// TwinCAT 3 PLC project PLC_Framework_V2_00
// ProgramVersion: 3.1.4023.0
// libraries:
//   CAA Memory, * (CAA Technical Workgroup)
//   Tc2_Math, * (Beckhoff Automation GmbH)
//   Tc2_MC2, * (Beckhoff Automation GmbH)
//   Tc2_MC2_Drive, * (Beckhoff Automation GmbH)
//   Tc2_Standard, * (Beckhoff Automation GmbH)
//   Tc2_System, * (Beckhoff Automation GmbH)
//   Tc2_Utilities, * (Beckhoff Automation GmbH)
//   Tc3_Module, * (Beckhoff Automation GmbH)
// project tree:
//   / CheckBounds.TcPOU, CheckDivDInt.TcPOU, CheckDivLInt.TcPOU, CheckDivLReal.TcPOU, CheckDivReal.TcPOU, CheckLRangeSigned.TcPOU, CheckLRangeUnsigned.TcPOU, CheckPointer.TcPOU, CheckRangeSigned.TcPOU, CheckRangeUnsigned.TcPOU, PlcTask.TcTTO
//   GVLs/ GVL_Module.TcGVL, GVL_Constant.TcGVL, GVL_Standard.TcGVL
//   POUs/ MAIN.TcPOU
//   Standard/ CallStandard.TcPOU, CallStandardModule.TcPOU
//   Standard/ENUM/ ENUM_CarrierPos.TcDUT, ENUM_ExecState.TcDUT, ENUM_NgReason.TcDUT, ENUM_ProductState.TcDUT, ENUM_StationCommand.TcDUT, ENUM_UnitState.TcDUT
//   Standard/FUN/ FUN_AryBitCount_RD.TcPOU, FUN_AryBitOnNum_RD.TcPOU, FUN_AryToLword_RD.TcPOU, FUN_AryToWord_RD.TcPOU, FUN_TimeToDate_RD.TcPOU, FUN_UpdateLeftSidebar_RD.TcPOU, FUN_WordToAry.TcPOU, F_Sum.TcPOU
//   Standard/Module/Connector/Termininal/ FB_Terminal2_RD.TcPOU, FB_Terminal_RD.TcPOU, UDT_TerminalData_RD.TcDUT, UDT_TerminalHmi_RD.TcDUT, UDT_TerminalMessage_RD.TcDUT, UDT_TerminalVar_RD.TcDUT, UDT_Terminal_RD.TcDUT
//   Standard/Module/FAKRA/BraidFlaring/ FB_BraidFlaring_RD.TcPOU, UDT_BraidFlaring_RD.TcDUT, UDT_Data_BraidFlaring_RD.TcDUT, UDT_Hmi_BraidFlaring_RD.TcDUT, UDT_Imm_BraidFlaring_RD.TcDUT, UDT_Parameters_BraidFlaring_RD.TcDUT
//   Standard/Module/FAKRA/Crimping/ FB_Crimping_RD.TcPOU, UDT_Crimping_RD.TcDUT, UDT_Data_Crimping_RD.TcDUT, UDT_Hmi_Crimping_RD.TcDUT, UDT_Imm_Crimping_RD.TcDUT, UDT_Parameters_Crimping_RD.TcDUT
//   Standard/Module/FAKRA/JacketStripping/ FB_JacketStripping_RD.TcPOU, UDT_CriticalProcessParameters_JacketStripping_RD.TcDUT, UDT_Data_JacketStripping_RD.TcDUT, UDT_Hmi_JacketStripping_RD.TcDUT, UDT_Imm_JacketStripping_RD.TcDUT, UDT_JacketStripping_RD.TcDUT
//   Standard/Public/00 System/ FB_Blinker_RD.TcPOU, FB_GetPlcClock.TcPOU, UDT_PlcStatus_RD.TcDUT, UDT_ProgramStatus_RD.TcDUT, UDT_System_RD.TcDUT
//   Standard/Public/01 Machine/ FB_Machine_RD.TcPOU, UDT_MachineHmi_RD.TcDUT, UDT_MachineReport_RD.TcDUT, UDT_MachineSidebar_RD.TcDUT, UDT_Machine_RD.TcDUT
//   Standard/Public/02 Station/ FB_Station_RD.TcPOU, UDT_FlowHmi_RD.TcDUT, UDT_Flow_RD.TcDUT, UDT_StationHmi_RD.TcDUT, UDT_StationMessage_RD.TcDUT, UDT_StationReport_RD.TcDUT, UDT_StationSidebar_RD.TcDUT, UDT_Station_RD.TcDUT
//   Standard/Public/03 HMI/ UDT_RightSidebar_RD.TcDUT, FB_GetPageSerialNo_RD.TcPOU, FB_GetPlcClock_RD.TcPOU, FB_Hmi_RD.TcPOU, FB_IV3_G120_RD.TcPOU, FB_Tben_L5_4Rfid_RD.TcPOU, FB_TurnPages_RD.TcPOU, FB_UpdateAxisHmi_RD.TcPOU, FB_UpdateCycleTimeHmi_RD.TcPOU, FB_UpdateInsertHmi_RD.TcPOU, FB_UpdateProduceHmi_RD.TcPOU, UDT_Clock_RD.TcDUT, UDT_CycleTimeHmi_RD.TcDUT, UDT_DayTime_RD.TcDUT, UDT_Hmi_RD.TcDUT, UDT_HmiButton_RD.TcDUT, UDT_LeftSidebar_RD.TcDUT, UDT_TurnPages_RD.TcDUT
//   Standard/Public/06 Produce/ FB_Produce_RD.TcPOU, FB_Produce.TcPOU, UDT_BadData_RD.TcDUT, UDT_BadHmi_RD.TcDUT, UDT_BadVar_RD.TcDUT, UDT_ProduceDataRecord_RD.TcDUT, UDT_ProduceData_RD.TcDUT, UDT_ProduceHmi_RD.TcDUT, UDT_ProduceVar_RD.TcDUT
//   Standard/Public/08 WearPart/ FB_WearPart.TcPOU, UDT_WearPartData_RD.TcDUT, UDT_WearPartHmi_RD.TcDUT, UDT_WearPartVar_RD.TcDUT
//   Standard/Public/11 Oee/ FB_Oee_RD.TcPOU, UDT_OeeData_RD.TcDUT, UDT_OeeHmi_RD.TcDUT, UDT_OeeVar_RD.TcDUT
//   Standard/Unit/00 General/ FB_Click_RD.TcPOU
//   Standard/Unit/03 Estop/ FB_Estop_RD.TcPOU, UDT_Estop_RD.TcDUT
//   Standard/Unit/04 SafetyDoor/ FB_SafetyDoor_RD.TcPOU, UDT_SafetyDoor_RD.TcDUT
//   Standard/Unit/05 Cylinder/ FB_Cylinder_RD.TcPOU, UDT_CylinderData_RD.TcDUT, UDT_CylinderHmi_RD.TcDUT, UDT_CylinderMessage_RD.TcDUT, UDT_CylinderVar_RD.TcDUT
//   Standard/Unit/06 Axis/ FB_Axis_RD.TcPOU, FB_ModuloCalculate_RD.TcPOU, FB_NCI.TcPOU, UDT_AxisData_RD.TcDUT, UDT_AxisHmi_RD.TcDUT, UDT_AxisMessage_RD.TcDUT, UDT_AxisVar_RD.TcDUT, UDT_ModuloProperty_RD.TcDUT
//   Standard/Unit/07 Sensor/ FB_Sensor_RD.TcPOU, UDT_SensorData_RD.TcDUT, UDT_SensorHmi_RD.TcDUT, UDT_SensorVar_RD.TcDUT
//   Standard/Unit/08 Motor/ FB_Motor_RD.TcPOU, UDT_MotorData_RD.TcDUT, UDT_MotorHmi_RD.TcDUT, UDT_MotorVar_RD.TcDUT
//   Standard/Unit/11 KeyenceScan/ FB_KeyenceScan_RD.TcPOU, UDT_KeyenceScanData_RD.TcDUT, UDT_KeyenceScanHmi_RD.TcDUT, UDT_KeyenceScanVar_RD.TcDUT
//   Standard/Unit/12 Delay/ FB_Delay_RD.TcPOU, UDT_DelayData_RD.TcDUT, UDT_DelayHmi_RD.TcDUT, UDT_DelayVar_RD.TcDUT
//   Standard/Unit/13 Valve/ FB_Valve_RD.TcPOU, UDT_ValveData_RD.TcDUT, UDT_ValveHmi_RD.TcDUT, UDT_ValveVar_RD.TcDUT
//   Standard/Unit/40 RackFeeder/ FB_RackFeeder_RD.TcPOU, UDT_RackFeederData_RD.TcDUT, UDT_RackFeederHmi_RD.TcDUT, UDT_RackFeederInput_RD.TcDUT, UDT_RackFeederOutput_RD.TcDUT, UDT_RackFeederVar_RD.TcDUT, UDT_RackFeedMessage_RD.TcDUT

CONFIGURATION PLC_Framework_V2_00
    RESOURCE PLC ON TwinCAT3
        TASK PlcTask(INTERVAL := T#10ms, PRIORITY := 20);
        PROGRAM MAIN WITH PlcTask : MAIN;
    END_RESOURCE
END_CONFIGURATION

// ---- Standard/ENUM/ENUM_CarrierPos.TcDUT
TYPE ENUM_CarrierPos :
(
	Left 	:= 1,
	Right 	:= 2
)UINT;
END_TYPE

// ---- Standard/ENUM/ENUM_ExecState.TcDUT
{attribute 'qualified_only'}
{attribute 'strict'}
TYPE ENUM_ExecState :
(
	NOT_READY := 1,
  READY :=2,
  RUNNING :=3,
  DONE :=4,
  CANCEL :=5,
  INIT := 6,
  ERROR :=7

);
END_TYPE

// ---- Standard/ENUM/ENUM_NgReason.TcDUT
{attribute 'qualified_only'}
{attribute 'strict'}
TYPE ENUM_NgReason :
(
	CrimpNoCable :=1,
	CrimpNg,
	CrimpInterrupted,
	LastReason
);
END_TYPE

// ---- Standard/ENUM/ENUM_ProductState.TcDUT
{attribute 'qualified_only'}
{attribute 'strict'}
TYPE ENUM_ProductState :
(
	Empty:=0,					//无产品
	Good:=1,					//良品
	Bad:=2,						//不良品
	New:=3,						//新产品
	Sample:=4					//送检样品
);
END_TYPE

// ---- Standard/ENUM/ENUM_StationCommand.TcDUT
{attribute 'qualified_only'}
{attribute 'strict'}
TYPE ENUM_StationCommand :
(
  	
    INIT :=1,
    START := 2,
    STOP :=3,
    PAUSE := 4
    
    
  
);
END_TYPE

// ---- Standard/ENUM/ENUM_UnitState.TcDUT
{attribute 'qualified_only'}
{attribute 'strict'}
TYPE ENUM_UnitState :
(
  
	DISABLED := 1,
  OPERATIONAL :=2,
  STANDBY :=3,
  UNKNOWN :=4

);
END_TYPE

// ---- Standard/Module/Connector/Termininal/UDT_TerminalData_RD.TcDUT
TYPE UDT_TerminalData_RD :
STRUCT
timeout           : TIME; //对端子超时
terminalSensor    : UDT_SensorData_RD; //端子有无感应
coverSensor       : UDT_SensorData_RD; //盖板感应
pinSensor         : UDT_SensorData_RD; //对Pin感应
END_STRUCT
END_TYPE

// ---- Standard/Module/Connector/Termininal/UDT_TerminalHmi_RD.TcDUT
TYPE UDT_TerminalHmi_RD :
STRUCT
terminalSensor    : UDT_SensorHmi_RD; //端子有无感应
coverSensor       : UDT_SensorHmi_RD; //盖板感应
pinSensor         : UDT_SensorHmi_RD; //对Pin感应
hmi               : BOOL; //对端子Hmi
manual            : BOOL; //对端子手动执行
forbidIcon        : BOOL; //禁止图标
display           : BOOL; //显示
ready             : BOOL; //对端子准备就绪
busy              : BOOL; //对端子中
done              : BOOL; //对端子完成
subDisplay        : BOOL; //子画面显示
number            : INT; //编号
flowStep          : INT; //流程步
status            : INT; //状态
timeout           : DINT; //对端子超时
END_STRUCT
END_TYPE

// ---- Standard/Module/Connector/Termininal/UDT_TerminalMessage_RD.TcDUT
TYPE UDT_TerminalMessage_RD :
STRUCT
timeoutAlarm       : BOOL; //对端子超时报警
lackTerminalAlarm  : BOOL; //缺端子报警
coverAlarm         : BOOL; //盖板未检测到报警
alarming           : BOOL; //报警
END_STRUCT
END_TYPE

// ---- Standard/Module/Connector/Termininal/UDT_TerminalVar_RD.TcDUT
TYPE UDT_TerminalVar_RD :
STRUCT
terminalSensor       : UDT_SensorVar_RD; //端子有无感应
coverSensor          : UDT_SensorVar_RD; //盖板感应
pinSensor            : UDT_SensorVar_RD; //对Pin感应
disable              : BOOL; //屏蔽
hmi                  : BOOL; //对端子Hmi
manual               : BOOL; //对端子手动执行
auto                 : BOOL; //对端子自动执行
forbidIcon           : BOOL; //禁止图标
camAxisEnable        : BOOL; //插针凸轮轴启用
cutEnable            : BOOL; //裁切端子启用
running              : BOOL; //对端子运行中
ready                : BOOL; //对端子准备就绪
busy                 : BOOL; //对端子中
permit               : BOOL; //对端子条件
allow                : BOOL; //对端子可动作
done                 : BOOL; //对端子完成
faile                : BOOL; //对端子失败
timeoutAlarm         : BOOL; //对端子超时报警
lackTerminalAlarm    : BOOL; //缺端子报警
coverAlarm           : BOOL; //盖板未检测到报警
lackTerminalAutoTip  : BOOL; //缺端子自动提示
coverAutoTip         : BOOL; //盖板未检测到自动提示
alarming             : BOOL; //报警中
manualTip            : BOOL; //手动提示
autoTip              : BOOL; //自动提示
flowStep             : UINT; //流程步
status               : UINT; //状态
camAxisNo            : UINT; //凸轮轴
sendAxisNo           : UINT; //送端子轴
stationNo            : UINT; //所属工站编号
serialNo             : UINT; //HMI显示序号
END_STRUCT
END_TYPE

// ---- Standard/Module/Connector/Termininal/UDT_Terminal_RD.TcDUT
TYPE UDT_Terminal_RD :
STRUCT
send1Finish     : BOOL; //上进端子完成
send2Finish     : BOOL; //下进端子完成
send1Auto       : BOOL; //上进端子自动
send2Auto       : BOOL; //下进端子自动
END_STRUCT
END_TYPE

// ---- Standard/Module/FAKRA/BraidFlaring/UDT_BraidFlaring_RD.TcDUT
TYPE UDT_BraidFlaring_RD :
STRUCT
  
Imm : UDT_Imm_BraidFlaring_RD;
Message : UDT_StationMessage_RD;
Hmi : UDT_Hmi_BraidFlaring_RD;

UnitState : INT;	//DISABLED := 1,OPERATIONAL :=2,STANDBY :=3,UNKNOWN :=4
Command :INT; //INIT :=1,START := 2,STOP :=3,PAUSE := 4
CommandState : INT ; 	//NOT_READY := 1,READY :=2,RUNNING :=3,DONE :=4,CANCEL :=5,INIT := 6,ERROR :=7

END_STRUCT
END_TYPE

// ---- Standard/Module/FAKRA/BraidFlaring/UDT_Data_BraidFlaring_RD.TcDUT
TYPE UDT_Data_BraidFlaring_RD :
STRUCT
  
  gripCyl:UDT_CylinderData_RD;
  jackCyl:UDT_CylinderData_RD;
  pushCyl:UDT_CylinderData_RD;
  fixCyl:UDT_CylinderData_RD;
  stepFixCyl:UDT_CylinderData_RD;
  blow:UDT_CylinderData_RD;
  vacuum:UDT_CylinderData_RD;
  
  transferAxis : UDT_AxisData_RD;
  rotateAxis : UDT_AxisData_RD; 
  
  badDetectData :UDT_BadData_RD;//1227
  
  CPP : UDT_Parameters_BraidFlaring_RD;

END_STRUCT
END_TYPE

// ---- Standard/Module/FAKRA/BraidFlaring/UDT_Hmi_BraidFlaring_RD.TcDUT
TYPE UDT_Hmi_BraidFlaring_RD :
STRUCT

gripCyl:UDT_CylinderHmi_RD;
jackCyl:UDT_CylinderHmi_RD;
pushCyl:UDT_CylinderHmi_RD;
fixCyl:UDT_CylinderHmi_RD;
stepFixCyl:UDT_CylinderHmi_RD;
blow:UDT_CylinderHmi_RD;
vacuum:UDT_CylinderHmi_RD;

transferAxis : UDT_AxisHmi_RD; 
rotateAxis : UDT_AxisHmi_RD;

badDetect:UDT_BadHmi_RD;// 1227

station : UDT_StationHmi_RD;

END_STRUCT
END_TYPE

// ---- Standard/Module/FAKRA/BraidFlaring/UDT_Imm_BraidFlaring_RD.TcDUT
TYPE UDT_Imm_BraidFlaring_RD :
STRUCT
  
//公共接口
 Machine_eStop : BOOL;
 Machine_safety : BOOL;
 Machine_airOn : BOOL;
 Machine_allDoorClosed : BOOL;
 Machine_manualMode : BOOL; 
 Machine_autoMode : BOOL;
 Machine_reset :BOOL;
 Machine_stopping :BOOL;
 Machine_paused: BOOL;
 Machine_running :BOOL;

 
 //模组参数输入
 
 carrierNum		: UINT;	//载座编号（INPUT）
 carrierInPos : BOOL; //载座到位（INPUT）
 carrierPos :UINT; //载座位置（左1/右2）（INPUT）
 carrierState:UINT;//载座状态    //1227
 stationCanRun :BOOL;//模组动作条件（INPUT）
 
 //模组参数输出
 stationDone :BOOL;//模组完成（OUTPUT）
 carrierFree :BOOL;//载座不干涉（OUTPUT）
 carrierLeftProductState :INT; //左载座产品状态（OUTPUT）
 carrierRightProductState :INT;//右载座产品状态（OUTPUT）
 allObjectInitPos:BOOL;//所有部件在初始位置（OUTPUT）

 
END_STRUCT
END_TYPE

// ---- Standard/Module/FAKRA/BraidFlaring/UDT_Parameters_BraidFlaring_RD.TcDUT
TYPE UDT_Parameters_BraidFlaring_RD :
STRUCT
	clipEnable						: ARRAY [1..5] OF BOOL;
	transferAxisClipPosOffset		: ARRAY [1..5] OF REAL;
	rotateAxisClipPosOffset		    : ARRAY [1..5] OF REAL;
	transferAxisPushStartPosOffset	: REAL;
	transferAxisPushEndPosOffset	: REAL;
	rotateAxisPushPosOffset		    : REAL;
	rotateAxisBasePos				: REAL;
	transferAxisBasePos			    : REAL;
	override :INT;
END_STRUCT
END_TYPE

// ---- Standard/Module/FAKRA/Crimping/UDT_Crimping_RD.TcDUT
TYPE UDT_Crimping_RD :
STRUCT
  
Imm : UDT_Imm_Crimping_RD;
Message : UDT_StationMessage_RD;
Hmi : UDT_Hmi_Crimping_RD;

UnitState : INT;	//DISABLED := 1,OPERATIONAL :=2,STANDBY :=3,UNKNOWN :=4
Command :INT; //INIT :=1,START := 2,STOP :=3,PAUSE := 4
CommandState : INT ; 	//NOT_READY := 1,READY :=2,RUNNING :=3,DONE :=4,CANCEL :=5,INIT := 6,ERROR :=7

END_STRUCT
END_TYPE

// ---- Standard/Module/FAKRA/Crimping/UDT_Data_Crimping_RD.TcDUT
TYPE UDT_Data_Crimping_RD :
STRUCT
  
  gripCyl:UDT_CylinderData_RD;
  jack1Cyl:UDT_CylinderData_RD;
  jack2Cyl:UDT_CylinderData_RD;
  cutCyl:UDT_CylinderData_RD;
  feedCyl:UDT_CylinderData_RD;
  changeCyl:UDT_CylinderData_RD;
  fixCyl:UDT_CylinderData_RD;
  stepFixCyl:UDT_CylinderData_RD;
  carrierHold1Cyl:UDT_CylinderData_RD;
  carrierHold2Cyl:UDT_CylinderData_RD;
  jack3Cyl:UDT_CylinderData_RD;
  blow:UDT_CylinderData_RD;
  
  transferAxis : UDT_AxisData_RD; 
  crimpAxis : UDT_AxisData_RD;  
  
  rackFeeder:UDT_RackFeederData_RD;
  
  produceData:UDT_ProduceData_RD;
  badData: ARRAY[0..ENUM_NgReason.CrimpNg] OF UDT_BadData_RD;
  lastProduce:UDT_ProduceDataRecord_RD;
  
  CPP : UDT_Parameters_Crimping_RD;
  
  wearPart1 : UDT_WearPartData_RD;
  wearPart2 : UDT_WearPartData_RD;
 
  cableCheckSensorDisabled            : BOOL;
  terminalCheckSensorDisabled         : BOOL;
  terminalReiveCheckSensorDisabled    : BOOL;
  crimpHomeCheckSensorDisabled        : BOOL;
  oesDisabled                         : BOOL;  
  
END_STRUCT
END_TYPE

// ---- Standard/Module/FAKRA/Crimping/UDT_Hmi_Crimping_RD.TcDUT
TYPE UDT_Hmi_Crimping_RD :
STRUCT

gripCyl:UDT_CylinderHmi_RD;
jack1Cyl:UDT_CylinderHmi_RD;
jack2Cyl:UDT_CylinderHmi_RD;
cutCyl:UDT_CylinderHmi_RD;
feedCyl:UDT_CylinderHmi_RD;
changeCyl:UDT_CylinderHmi_RD;
fixCyl:UDT_CylinderHmi_RD;
stepFixCyl:UDT_CylinderHmi_RD;
carrierHold1Cyl:UDT_CylinderHmi_RD;
carrierHold2Cyl:UDT_CylinderHmi_RD;  
jack3Cyl:UDT_CylinderHmi_RD;
blow:UDT_CylinderHmi_RD; 

transferAxis : UDT_AxisHmi_RD; 
crimpAxis : UDT_AxisHmi_RD;

rackFeeder:UDT_RackFeederHmi_RD;

bad:UDT_BadHmi_RD;
produce:UDT_ProduceHmi_RD;

station : UDT_StationHmi_RD;

END_STRUCT
END_TYPE

// ---- Standard/Module/FAKRA/Crimping/UDT_Imm_Crimping_RD.TcDUT
TYPE UDT_Imm_Crimping_RD :
STRUCT
  
//公共接口
 Machine_eStop : BOOL;
 Machine_safety : BOOL;
 Machine_airOn : BOOL;
 Machine_allDoorClosed : BOOL;
 Machine_manualMode : BOOL; 
 Machine_autoMode : BOOL;
 Machine_reset :BOOL;
 Machine_stopping :BOOL;
 Machine_paused: BOOL;
 Machine_running :BOOL;

 
 //模组参数输入
 
 carrierNum		: UINT;	//载座编号（INPUT）
 carrierInPos : BOOL; //载座到位（INPUT）
 carrierPos :UINT; //载座位置（左1/右2）（INPUT）
 carrierState:UINT;//载座状态    //1227
 stationCanRun :BOOL;//模组动作条件（INPUT）
 
 //模组参数输出
 stationDone :BOOL;//模组完成（OUTPUT）
 carrierFree :BOOL;//载座不干涉（OUTPUT）
 carrierLeftProductState :INT; //左载座产品状态（OUTPUT）
 carrierRightProductState :INT;//右载座产品状态（OUTPUT）
 allObjectInitPos:BOOL;//所有部件在初始位置（OUTPUT）

 
END_STRUCT
END_TYPE

// ---- Standard/Module/FAKRA/Crimping/UDT_Parameters_Crimping_RD.TcDUT
TYPE UDT_Parameters_Crimping_RD :
STRUCT
	override :INT;
END_STRUCT
END_TYPE

// ---- Standard/Module/FAKRA/JacketStripping/UDT_CriticalProcessParameters_JacketStripping_RD.TcDUT
TYPE UDT_CriticalProcessParameters_JacketStripping_RD :
STRUCT
  
  blowTime :UDINT;
  firstCutTime :UDINT;
  firstOpenTime :UDINT;
  SecondCutTime :UDINT;
  secondOpenTime:UDINT;
  secondCutEnable	:BOOL;
  thirdCutTime	:UDINT;
  thirdOpenTime	:UDINT;
  thirdCutEnable	:BOOL;
  fourthCutTime	:UDINT;
  fourthOpenTime:	UDINT;
  fourthCutEnable	:BOOL;
  fifthCutTime	:UDINT;
  fifthOpenTime	:UDINT;
  fifthCutEnable	:BOOL;
  override :INT;
  
END_STRUCT
END_TYPE

// ---- Standard/Module/FAKRA/JacketStripping/UDT_Data_JacketStripping_RD.TcDUT
TYPE UDT_Data_JacketStripping_RD :
STRUCT
  
  gripCyl:UDT_CylinderData_RD;
  jackCyl:UDT_CylinderData_RD;
  fixCyl:UDT_CylinderData_RD;
  stepFixCyl:UDT_CylinderData_RD;
  blow:UDT_CylinderData_RD; 
  
  transferAxis : UDT_AxisData_RD; 
  cutAxis : UDT_AxisData_RD;  
  rotateAxis : UDT_AxisData_RD; 
  
  CPP : UDT_CriticalProcessParameters_JacketStripping_RD;
  
  wearPart : UDT_WearPartData_RD;
 
  
  
END_STRUCT
END_TYPE

// ---- Standard/Module/FAKRA/JacketStripping/UDT_Hmi_JacketStripping_RD.TcDUT
TYPE UDT_Hmi_JacketStripping_RD :
STRUCT
  
gripCyl : UDT_CylinderHmi_RD;
jackCyl :UDT_CylinderHmi_RD;
fixCyl  :UDT_CylinderHmi_RD;
stepFixCyl:UDT_CylinderHmi_RD; 
blow    :UDT_CylinderHmi_RD;

rotateAxis : UDT_AxisHmi_RD; 
cutAxis : UDT_AxisHmi_RD; 
transferAxis : UDT_AxisHmi_RD;

station : UDT_StationHmi_RD;

END_STRUCT
END_TYPE

// ---- Standard/Module/FAKRA/JacketStripping/UDT_Imm_JacketStripping_RD.TcDUT
TYPE UDT_Imm_JacketStripping_RD :
STRUCT
  
//公共接口（由外部机台输入）
 machine_eStop : BOOL;
 machine_safety : BOOL;
 machine_airOn : BOOL;
 machine_allDoorClosed : BOOL;
 machine_manualMode : BOOL; 
 machine_autoMode : BOOL;
 
 machine_running :BOOL;
 machine_stopping :BOOL;
 machine_initing :BOOL;
 machine_pause :BOOL;
 machine_reset :BOOL;

 //模组参数输入
 
 carrierNum		: UINT;	//载座编号（INPUT）
 carrierInPos : BOOL; //载座到位（INPUT）
 carrierPos :UINT; //载座位置（左1/右2）（INPUT）
 stationCanRun :BOOL;//模组动作条件（INPUT）

 
 //模组参数输出
 
 stationAlarming :BOOL;//模组报警中（OUTPUT）
 stationRunning :BOOL;//模组运行中（OUTPUT）
 stationInitDone :BOOL;//模组初始化完成（Output）
 stationDone :BOOL;//模组完成（OUTPUT）
 carrierFree :BOOL;//载座不干涉（OUTPUT）
 carrierLeftProductState :INT; //左载座产品状态（OUTPUT）
 carrierRightProductState :INT;//右载座产品状态（OUTPUT）
 allObjectInitPos:BOOL;//所有部件在初始位置（OUTPUT）
 
END_STRUCT
END_TYPE

// ---- Standard/Module/FAKRA/JacketStripping/UDT_JacketStripping_RD.TcDUT
TYPE UDT_JacketStripping_RD :
STRUCT
  
Imm : UDT_Imm_JacketStripping_RD;
Message : UDT_StationMessage_RD;
Hmi : UDT_Hmi_JacketStripping_RD;

UnitState : INT;	//DISABLED := 1,OPERATIONAL :=2,STANDBY :=3,UNKNOWN :=4
Command :INT; //INIT :=1,START := 2,STOP :=3,PAUSE := 4
CommandState : INT ; 	//NOT_READY := 1,READY :=2,RUNNING :=3,DONE :=4,CANCEL :=5,INIT := 6,ERROR :=7


END_STRUCT
END_TYPE

// ---- Standard/Public/00 System/UDT_PlcStatus_RD.TcDUT
TYPE UDT_PlcStatus_RD :
STRUCT
  
cycleTime : TIME; // 周期时间
maxCycleTime : Time; // 最长循环时间
minCycleTime : Time; // 最短循环时间
systemClock : DATE_AND_TIME; // 系统时钟
localClock : DATE_AND_TIME; // 本地时钟
status : Int; // CPU运行状态

END_STRUCT
END_TYPE

// ---- Standard/Public/00 System/UDT_ProgramStatus_RD.TcDUT
TYPE UDT_ProgramStatus_RD :
STRUCT
 
error : BOOL; // 有错误
errorID : Word; // 错误代码
errorText : String[100]; // 错误文本信息
warning : Bool; // 有警告
warnID : Word; // 警告代码
warnText : String[100]; // 警告文本信息
  
END_STRUCT
END_TYPE

// ---- Standard/Public/00 System/UDT_System_RD.TcDUT
TYPE UDT_System_RD :
STRUCT
clock	: UDT_Clock_RD;
plcStatus :	UDT_PlcStatus_RD;				
programStatus	: UDT_ProgramStatus_RD;
 
END_STRUCT
END_TYPE

// ---- Standard/Public/01 Machine/UDT_MachineHmi_RD.TcDUT
TYPE UDT_MachineHmi_RD :
STRUCT
eStop : BOOL; //急停
airOn : BOOL; //气压
allDoorClosed : BOOL; //安全门
ready : Bool; //准备就绪
running : Bool; //运行中
alarming : Bool; //报警中
paused : Bool; //暂停中
stopping : Bool; //停止中
tipReset : Bool; // 提示复位
initConfirm : Bool; // 整机初始化确认
emptyConfirm : Bool; // 清料确认
emptyhmi : Bool; // 清料hmi
emptying : Bool; // 清料中
emptyDone : Bool; // 清料完成
dummying : Bool; // 点检中
dummyDone : Bool; // 点检完成
dryRun : Bool; // 空跑
startButtonLight : Bool; // 启动按钮指示灯
stopButtonLight : Bool; // 停止按钮指示灯
resetButtonLight : Bool; // 复位按钮指示灯
pauseButtonLight : Bool; // 暂停按钮指示灯
initButtonLight : Bool; // 初始化按钮指示灯
starthmi : Bool; // 启动hmi
stophmi : Bool; // 停止hmi
resethmi : Bool; // 复位hmi
pausehmi : Bool; // 暂停hmi
inithmi : Bool; // 整机初始化hmi
manualModehmi : Bool; // 手动模式hmi
autoModehmi : Bool; // 自动模式hmi
jogModehmi : Bool; // 寸动模式hmi
setupModehmi : Bool; // 调试模式hmi
lampTesthmi : Bool; // 指示灯测试hmi
floodlighthmi : Bool; // 照明灯光打开hmi
alarmTopBarDisplay : Bool; // 报警顶栏显示
actAlarmTimes : UInt; // 当前发生报警条数
status : UInt; // 整机状态显示
initStatus : UInt; // 整机初始化状态显示
mode : UInt; // 操作模式
haveControlhmiNo : Int; // 当前拥有该机器控制权的hmi编号
requestControlhmiNo : Int; // 请求该机器控制权的hmi编号
requestCountdown : Int; // hmi请求控制权倒计时
actLanguage : Int; // 当前使用语言
mainScreenNo : Int; // 主画面编号
popup : Int; // 触摸屏弹窗
flow : Array[0..7] of UDT_FlowHmi_RD; // 流程
sidebar : UDT_LeftSidebar_RD; //
number : Int; // 机器编号
  
END_STRUCT
END_TYPE

// ---- Standard/Public/01 Machine/UDT_MachineReport_RD.TcDUT
TYPE UDT_MachineReport_RD :
STRUCT
alarming : BOOL; // 其它报警中
manualTip : Bool; // 其它手动提示
autoTip : Bool; // 其它自动提示
alarmCanReset : Bool; // 报警可复位
notSafetyDoors : Bool; // 安全门未就绪
notEstops : Bool; // 急停未就绪
stationAlarming : Bool; // 工站报警中
stationManualTip : Bool; // 工站手动提示
stationAutoTip : Bool; // 工站自动提示
stationNotInitDone : Bool; // 工站初始化未完成

END_STRUCT
END_TYPE

// ---- Standard/Public/01 Machine/UDT_MachineSidebar_RD.TcDUT
TYPE UDT_MachineSidebar_RD :
STRUCT
typeData : ARRAY[0..31] OF INT; // 按钮类型
status : ARRAY[0..31] OF Bool; // 按钮状态
click : ARRAY[0..31] OF Bool; // 按钮操作 
END_STRUCT
END_TYPE

// ---- Standard/Public/01 Machine/UDT_Machine_RD.TcDUT
TYPE UDT_Machine_RD :
STRUCT
startUp : BOOL; // 上电或切换语言
eStop : Bool; // 急停
safety : Bool; // 安全防护
airOn : Bool; // 气压正常
allDoorClosed : Bool; // 所有安全门关好
ready : Bool; // 准备就绪
start : Bool; // 启动
stop : Bool; // 停止
reset : Bool; // 复位
pause : Bool; // 暂停
init : Bool; // 初始化
manualMode : Bool; // 手动模式
autoMode : Bool; // 自动模式
jogMode : Bool; // 寸动模式
setupMode : BOOL; // 调试模式
releaseMode : BOOL; //抽检模式
tipReset : Bool; // 提示复位
running : Bool; // 运行中
stopping : Bool; // 停止中
stopDoneAllow : Bool; // 停止完成允许
stopDone : Bool; // 停止完成
alarming : Bool; // 机器报警中
paused : Bool; // 暂停中
initConfirm : Bool; // 整机初始化确认
initing : Bool; // 整机初始化中
initDone : Bool; // 整机初始化完成
initDelay : Bool; // 整机初始化延时
initFlowDone : Bool; // 整机初始化流程结束
emptyConfirm : Bool; // 清料确认
emptyhmi : Bool; // 清料hmi
emptying : Bool; // 清料中
emptyDone : Bool; // 清料完成
dummying : Bool; // 点检中
dummyDone : Bool; // 点检完成
manualTip : Bool; // 手动提示中
autoTip : Bool; // 自动提示中
autoTipTrigger : Bool; // 自动提示触发显示
publicAlarm : Bool; // 公共报警中
alarmCanReset : Bool; // 报警可复位
dryRun : Bool; // 空跑
runPermit : Bool; // 机器运行条件
startPermit : Bool; // 启动条件
startButton : Bool; // 启动按钮
stopButton : Bool; // 停止按钮
resetButton : Bool; // 复位按钮
pauseButton : Bool; // 暂停按钮
initButton : Bool; // 初始化按钮
manualSwitch : Bool; // 手动模式开关
autoSwitch : Bool; // 自动模式开关
startButtonLight : Bool; // 启动按钮指示灯
stopButtonLight : Bool; // 停止按钮指示灯
resetButtonLight : Bool; // 复位按钮指示灯
pauseButtonLight : Bool; // 暂停按钮指示灯
initButtonLight : Bool; // 初始化按钮指示灯
redStatusLight : Bool; // 三色灯红
yellowStatusLight : Bool; // 三色灯黄
greenStatusLight : Bool; // 三色灯绿
buzzer : Bool; // 三色灯蜂鸣器
starthmi : Bool; // 启动hmi
stophmi : Bool; // 停止hmi
resethmi : Bool; // 复位hmi
pausehmi : Bool; // 暂停hmi
inithmi : Bool; // 整机初始化hmi
manualModehmi : Bool; // 手动模式hmi
autoModehmi : Bool; // 自动模式hmi
jogModehmi : Bool; // 寸动模式hmi
setupModehmi : Bool; // 调试模式hmi
lampTesthmi : Bool; // 指示灯测试hmi
floodlighthmi : Bool; // 照明灯光打开hmi
alarmTopBarDisplay : Bool; // 报警顶栏显示
cycleTimeStart : Bool; // 机器周期计时开始
cycleTimeEnd : Bool; // 机器周期计时结束
cycleTime : DINT; // 机器周期时间
idealCycleTime : Time; // 机器理想周期时间
initTimeout : Time; // 初始化超时时间
stopTimeout : Time; // 停止超时时间
buzzerTime : Time; // 蜂鸣器持续时间
alarmCount : UInt; // 报警计数
actAlarmTimes : UInt; // 当前发生报警条数
status : UInt; // 整机状态显示
initStatus : UInt; // 整机初始化状态显示
mode : UInt; // 操作模式
haveControlhmiNo : UINT; // 当前拥有该机器控制权的hmi编号
requestControlhmiNo : UINT; // 请求该机器控制权的hmi编号
requestCountdown : UINT; // hmi请求控制权倒计时
actLanguage : UINT; // 当前使用语言
mainScreenNo : UINT; // 主画面编号
popup : UINT; // 触摸屏弹窗
machineNo : UINT; // 当前机器编号
flow : Array[0..5] of UDT_Flow_RD; // 流程
presetAlarms : Array[0..15] of Bool; // 预置报警
presetManualTips : Array[0..15] of Bool; // 预置手动提示
presetAutoTips : Array[0..15] of Bool; // 预置自动提示
presetTips : Array[0..31] of Bool; // 预置一般提示
userAlarms : Array[0..63] of Bool; // 用户报警
userManualTips : Array[0..63] of Bool; // 用户手动提示
userAutoTips : Array[0..63] of Bool; // 用户自动提示
userTips : Array[0..63] of Bool; // 用户一般提示
report : UDT_MachineReport_RD; // 下属状态反馈
sidebar : UDT_MachineSidebar_RD; // 左侧边栏



END_STRUCT
END_TYPE

// ---- Standard/Public/02 Station/UDT_FlowHmi_RD.TcDUT
TYPE UDT_FlowHmi_RD :
STRUCT
  
actStep : UINT; // 当前步号
number : INT; // 流程文本列表编号
name : STRING[20]; // 流程名称
describe : STRING[60]; // 流程说明
  
END_STRUCT
END_TYPE

// ---- Standard/Public/02 Station/UDT_Flow_RD.TcDUT
TYPE UDT_Flow_RD :
STRUCT
timeoutEnable : BOOL; // 超时检测开启
timeoutAlarm : Bool; // 超时报警输出
timeoutException : Bool; // 超时例外输入
uninterrupted : Bool; // 不停顿
setTimeout : Time; // 超时时间设置
prevStep : UInt; // 上一步号
nextStep : UInt; // 下一步号
actStep : UINT; // 当前步号
name : STRING[20]; // 流程名称
describe : STRING[60]; // 流程说明



END_STRUCT
END_TYPE

// ---- Standard/Public/02 Station/UDT_StationHmi_RD.TcDUT
TYPE UDT_StationHmi_RD :
STRUCT
inithmi : BOOL; // 工站初始化hmi
initForbidIcon : Bool; // 工站初始化禁止图标
initing : Bool; // 工站初始化中
cycleRunhmi : Bool; // 工站单循环hmi
cycleRunForbidIcon : Bool; // 工站单循环禁止图标
cycleRunning : Bool; // 工站单循环中
jogRunhmi : Bool; // 工站寸动hmi
jogRunForbidIcon : Bool; // 工站寸动禁止图标
jogRunning : Bool; // 工站寸动中
pausehmi : Bool; // 工站暂停hmi
disablehmi : Bool; // 工站屏蔽hmi
repetitionsEnable : Bool; // 单循环重复动作开启
repetitionsClear : Bool; // 单循环重复动作计数清零
repetitions : UInt; // 单循环重复动作计数
repetitionsTimes : UInt; // 单循环重复动作次数设置
status : UINT; // 工站状态显示 0工站报警中... 1工站未准备好 2工站准备好 3工站运行中 4工站单循环中 5工站单循环暂停中 6工站初始化中 7工站未初始化
flowDisplay : UInt; // 流程显示数量
flow : Array[0..5] of UDT_FlowHmi_RD; // 流程
number : INT; // 部件编号
selectPageValue : ARRAY[0..8] OF Int; // 工站选择页值
cycleTime : UDINT; // 工站周期时间
historicalCycleTime : ARRAY[1..5] OF UDINT; // 工站周期时间

END_STRUCT
END_TYPE

// ---- Standard/Public/02 Station/UDT_StationMessage_RD.TcDUT
TYPE UDT_StationMessage_RD :
STRUCT
presetAlarms : ARRAY[0..15] OF BOOL; // 预置报警
presetManualTips : Array[0..15] of Bool; // 预置手动提示
presetAutoTips : Array[0..15] of Bool; // 预置自动提示
userAlarms : Array[0..63] of Bool; // 用户报警
userManualTips : Array[0..63] of Bool; // 用户手动提示
userAutoTips : Array[0..63] of Bool; // 用户自动提示
userTips : ARRAY[0..63] OF BOOL; // 用户一般提示

presetAlarms16 : WORD;
presetManualTips16 : WORD;
presetAutoTips16: WORD;
userAlarms64 : LWORD;
userManualTips64 : LWORD;
userAutoTips64 : LWORD;
userTips64 : LWORD;

popupTrigger: WORD;

END_STRUCT
END_TYPE

// ---- Standard/Public/02 Station/UDT_StationReport_RD.TcDUT
TYPE UDT_StationReport_RD :
STRUCT
  
alarming : BOOL; // 其它报警中
manualTip : Bool; // 其它手动提示
autoTip : Bool; // 其它自动提示
  
END_STRUCT
END_TYPE

// ---- Standard/Public/02 Station/UDT_StationSidebar_RD.TcDUT
TYPE UDT_StationSidebar_RD :
STRUCT
otherEnable : BOOL; // 其它按钮启用
other2Enable : Bool; // 其它2按钮启用
other3Enable : Bool; // 其它3按钮启用
other4Enable : Bool; // 其它4按钮启用
otherIcon : Int; // 其它按钮图标编号
other2Icon : Int; // 其它2按钮图标编号
other3Icon : Int; // 其它3按钮图标编号
other4Icon : Int; // 其它4按钮图标编号
  
END_STRUCT
END_TYPE

// ---- Standard/Public/02 Station/UDT_Station_RD.TcDUT
TYPE UDT_Station_RD :
STRUCT
canRun : BOOL; // 工站可动作
inithmi : Bool; // 工站初始化hmi
initAllow : Bool; // 工站初始化允许操作
initAuto : Bool; // 工站初始化Auto
initForbidIcon : Bool; // 工站初始化禁止图标
initPermit : Bool; // 工站初始化条件
initing : Bool; // 工站初始化中
initDelay : Bool; // 工站初始化延时
initDone : Bool; // 工站初始化完成
cycleRunhmi : Bool; // 工站单循环hmi
cycleRunAllow : Bool; // 工站单循环允许操作
cycleRunAuto : Bool; // 工站单循环Auto
cycleRunForbidIcon : Bool; // 工站单循环禁止图标
cycleRunPermit : Bool; // 工站单循环条件
cycleRunning : Bool; // 工站单循环中
cycleRunFlag : Bool; // 工站单循环标志
jogRunhmi : Bool; // 工站寸动hmi
jogRunAllow : Bool; // 工站寸动允许操作
jogRunAuto : Bool; // 工站寸动Auto
jogRunForbidIcon : Bool; // 工站寸动禁止图标
jogRunPermit : Bool; // 工站寸动条件
jogRunning : Bool; // 工站寸动中
pausehmi : Bool; // 工站暂停hmi
disablehmi : Bool; // 工站屏蔽hmi
disablePermit : Bool; // 工站屏蔽条件
disabled : Bool; // 工站屏蔽中
ready : Bool; // 工站准备就绪
alarming : Bool; // 工站报警中
autoTip : Bool; // 工站自动提示中
autoTipTrigger : Bool; // 工站自动提示触发显示
manualTip : Bool; // 工站手动提示中
running : Bool; // 工站运行中
runPermit : Bool; // 工站运行条件
done : Bool; // 工站完成信号
cycleTimeStart : Bool; // 工站周期计时开始
cycleTimeEnd : Bool; // 工站周期计时结束
recordCycleTimeStart : Bool; // 工站详细周期计时开始
recordCycleTimeEnd : Bool; // 工站详细周期计时结束
requiresReinitialize : Bool; // 急停后工站需要重新初始化
syncAlarms : Bool; // 同步报警,其它工站报警本站立即停止
initResetAutoFlow : Bool; // 初始化时自动复位工站所有流程步
initSyncMachine : Bool; // 同步机器初始化，1:机器初始化中时单工站同步初始化
repetitionsEnable : Bool; // 单循环重复动作开启
sidebar : UDT_StationSidebar_RD; //
machineNo : UINT; // 所属机器编号
stationNo : UINT; // 当前工站编号
cycleTime : DINT; // 工站周期时间
initTimeout : Time; // 初始化超时时间
repetitions : UInt; // 单循环重复动作计数
repetitionsTimes : UInt; // 单循环重复动作次数设置
status : UInt; // 工站状态显示
flowDisplay : UINT; // 流程显示数量
flow : Array[0..5] of UDT_Flow_RD; // 流程
presetAlarms : Array[0..15] of Bool; // 预置报警
presetManualTips : Array[0..15] of Bool; // 预置手动提示
presetAutoTips : Array[0..15] of Bool; // 预置自动提示
userAlarms : Array[0..63] of Bool; // 用户报警
userManualTips : Array[0..63] of Bool; // 用户手动提示
userAutoTips : Array[0..63] of Bool; // 用户自动提示
userTips : Array[0..63] of Bool; // 用户一般提示
headerText : STRING[50]; // 标头文本
report : UDT_StationReport_RD; // 下级状态反馈
name : STRING[30]; // 工站名称

repetitionsClear : BOOL; // 单循环重复动作计数清零
  
END_STRUCT
END_TYPE

// ---- Standard/Public/03 HMI/UDT_RightSidebar_RD.TcDUT
TYPE UDT_RightSidebar_RD :
STRUCT
typeData : ARRAY[0..100] OF INT; // 按钮类型缓存
typeShow : Array[0..6] of Int; // 按钮类型显示
iconShow : Array[0..6] of Int; // 图标显示编号
textShow : Array[0..6] of Int; // 文本显示控制
buttonClick : Array[0..6] of bool; // 按钮点击
buttonStatus : Array[0..6] of bool; // 按钮状态
buttonClickNo : Int; // 按钮点击编号
pageUp : Bool; // 上一页按钮
pageDown : Bool; // 下一页按钮
pageUpDisplay : Bool; // 上一页按钮显示
pageDownDisplay : Bool; // 下一页按钮显示
 
END_STRUCT
END_TYPE

// ---- Standard/Public/03 HMI/UDT_Clock_RD.TcDUT
TYPE UDT_Clock_RD :
STRUCT
c1ms : BOOL; // 1ms时钟周期
c10ms : Bool; // 10ms时钟周期
c20ms : Bool; // 20ms时钟周期
c100ms : Bool; // 100ms时钟周期
c200ms : Bool; // 200ms时钟周期
c1s : Bool; // 1s时钟周期
c1min : Bool; // 1min时钟周期
p1ms : Bool; // 1ms时钟脉冲
p10ms : Bool; // 10ms时钟脉冲
p20ms : Bool; // 20ms时钟脉冲
p100ms : Bool; // 100ms时钟脉冲
p200ms : Bool; // 200ms时钟脉冲
p1s : Bool; // 1s时钟脉冲
p1min : Bool; // 1min时钟脉冲
p1hour : Bool; // 1hour时钟脉冲
  
END_STRUCT
END_TYPE

// ---- Standard/Public/03 HMI/UDT_CycleTimeHmi_RD.TcDUT
TYPE UDT_CycleTimeHmi_RD :
STRUCT
turnPages : UDT_TurnPages_RD; //
cycleTimeMax : Dint; // 周期时间MAX
cycleTimeMin : Dint; // 周期时间MIN
idealCycleTime : Dint; // 理想周期时间
number : Array[0..8] of int; // 编号
cycleTime : Array[0..8] of Dint; // 周期时间
display : Array[0..8] of Bool; // 工站显示
  
END_STRUCT
END_TYPE

// ---- Standard/Public/03 HMI/UDT_DayTime_RD.TcDUT
TYPE UDT_DayTime_RD :
STRUCT
times : TIME; // 总时间
timeValue :UDINT; //时间数值
day : USInt; // 天
hour : USInt; // 时
minute : USInt; // 分
second : USInt; // 秒

END_STRUCT
END_TYPE

// ---- Standard/Public/03 HMI/UDT_Hmi_RD.TcDUT
TYPE UDT_Hmi_RD :
STRUCT
changeDisplay : BOOL; // 切换机器按钮显示
nextPage : Bool; // 下一页按钮
prevPage : Bool; // 上一页按钮
nextPageDisplay : Bool; // 下一页按钮显示
prevPageDisplay : Bool; // 上一页按钮显示
nextStation : Bool; // 下一工站按钮
prevStation : Bool; // 上一工站按钮
nextStationDisplay : Bool; // 下一工站按钮显示
prevStationDisplay : Bool; // 上一工站按钮显示
requestControl : Bool; // hmi请求控制权
haveControl : Bool; // hmi拥有控制权
noControl : Bool; // hmi无控制权
selectMachineConfirm : Bool; // 选择机器编号确认
selectMachineTip : Bool; // 不能切换机器编号提示
requestCancel : Bool; // hmi请求控制权取消
requestConfirm : Bool; // hmi请求控制权确认
requestPopup : Bool; // hmi请求控制权弹窗
selectMachineNo : UINT; // 选择机器编号
machineNo : UINT; // 当前机器编号
stationNo : UINT; // 当前工站编号
stationIndex : UINT; // 当前工站索引下标
inputIndex : UINT; // IO检查Input索引
outputIndex : UINT; // IO检查Output索引
hmiNo : UINT; // hmi编号
hmiType : UINT; // hmi型号 0: TP700/900 1:TP1200/1500 2:TP1900 3:TP2200
language : UINT; // 语言选择
stationListValue : ARRAY[0..8] OF UINT; // 工站选择页值
stationListDisplay : BOOL; // 工站选择页显示
toManualPageClick : BOOL; //
toParameterPageClick : BOOL; //
toStationPageClick : BOOL; //
inManualPage : BOOL; //
inParameterPage : BOOL; //
inStationPage : BOOL; //
inOtherPage : BOOL; //
mainListDisplay : BOOL; //
statisticsListDisplay : BOOL; //
dummyCheckListDisplay : BOOL; //
ioCheckListDisplay : BOOL; //
helpListDisplay : BOOL; //
mainListShow : Int; //
statisticsListShow : UINT; //
dummyCheckListShow : UINT; //
ioCheckListShow : UINT; //
helpListShow : UINT; //
writePlcClockConfirm : BOOL; // 写入PLC时钟确认
writePlcClock : ARRAY[0..6] OF UINT; // 写入PLC时钟
readPlcClock : ARRAY[0..6] OF UINT; // 当前PLC时钟
leftSidebar : UDT_LeftSidebar_RD; // 左侧边栏
rightSidebar : UDT_RightSidebar_RD; // 右侧边栏
actPageNo : UINT; // 当前画面编号
pageUnitNo : ARRAY[0..8] OF UINT; // 当前画面显示部件编号
hmiControlWord : ARRAY[0..4] OF UINT; // hmi控制字
hmiPopupWord : ARRAY[0..3] OF UINT; // hmi弹窗控制字
machineName : STRING[20]; // 机器名称
canConnectMachine : Array[0..4] of Bool; // 可以连接机器
includingStationNum : Int; // 下属工站数量
includingStationIndex : ARRAY[0..50] OF UINT; // 下属工站索引下标
button : UDT_HmiButton_RD; // 按钮控制
machineHmi : UDT_MachineHmi_RD; //
stationHmi : UDT_StationHmi_RD; //
cycleTimeHmi : UDT_CycleTimeHmi_RD; //
cylinderHmi : ARRAY[1..8] OF UDT_CylinderHmi_RD; //
axisHmi : ARRAY[1..2] OF UDT_AxisHmi_RD; //
sensorHmi : ARRAY[1..8] OF UDT_SensorHmi_RD; //
motorHmi : ARRAY[1..8] OF UDT_MotorHmi_RD; //
delayHmi : ARRAY[1..8] OF UDT_DelayHmi_RD; //
valveHmi : ARRAY[1..8] OF UDT_ValveHmi_RD; //
rackFeederHmi : ARRAY[1..4] OF UDT_RackFeederHmi_RD; //
//bowlFeederHmi : ARRAY[1..2] OF UDT_BowlFeederHmi_RD; //
keyenceScanHmi : ARRAY[1..2] OF UDT_KeyenceScanHmi_RD; //
TerminalHmi : ARRAY[1..2] OF UDT_TerminalHmi_RD; //
produceHmi : UDT_ProduceHmi_RD; //
oeeHmi : UDT_OeeHmi_RD; //
//insertHmi : UDT_InsertHmi_RD; //
  
END_STRUCT
END_TYPE

// ---- Standard/Public/03 HMI/UDT_HmiButton_RD.TcDUT
TYPE UDT_HmiButton_RD :
STRUCT
start : BOOL; // 启动按钮
stop : Bool; // 停止按钮
reset : Bool; // 复位按钮
pause : Bool; // 暂停按钮
init : Bool; // 初始化按钮
manualSwitch : Bool; // 手动模式开关
autoSwitch : Bool; // 自动模式开关
startLight : Bool; // 启动按钮指示灯
stopLight : Bool; // 停止按钮指示灯
resetLight : Bool; // 复位按钮指示灯
pauseLight : Bool; // 暂停按钮指示灯
initLight : Bool; // 初始化按钮指示灯
  
END_STRUCT
END_TYPE

// ---- Standard/Public/03 HMI/UDT_LeftSidebar_RD.TcDUT
TYPE UDT_LeftSidebar_RD :
STRUCT
typeShow          : ARRAY[0..6] OF INT; // 按钮类型显示
StatusShow        : ARRAY[0..6] OF BOOL;// 按钮状态显示 1:ON 2:OFF
clickShow         : ARRAY[0..6] OF BOOL;// 按钮点击
pageUp            : BOOL;// 上一页按钮
pageDown          : BOOL;// 下一页按钮
pageUpDisplay     : BOOL;// 上一页按钮显示
pageDownDisplay   : BOOL;// 下一页按钮显示
END_STRUCT
END_TYPE

// ---- Standard/Public/03 HMI/UDT_TurnPages_RD.TcDUT
TYPE UDT_TurnPages_RD :
STRUCT
  
value : INT; // 页当前值
maxValue : Int; // 翻页最大值
minValue : Int; // 翻页最小值
increment : Int; // 单次增/减量
pageNumberDisplay : WORD; // 页码显示
prevDisplay : Bool; // 上一页按钮显示
nextDisplay : Bool; // 下一页按钮显示
prevClick : Bool; // 上一页按钮点击
nextClick : Bool; // 下一页按钮点击
 
END_STRUCT
END_TYPE

// ---- Standard/Public/06 Produce/UDT_BadData_RD.TcDUT
TYPE UDT_BadData_RD :
STRUCT
continuous : DINT; // 连续不良报警数量
cumulative : DInt; // 累计不良报警数量n
cumulativeRange : DInt; // 累计不良计算范围m
quantity : DInt; // 不良品数量

END_STRUCT
END_TYPE

// ---- Standard/Public/06 Produce/UDT_BadHmi_RD.TcDUT
TYPE UDT_BadHmi_RD :
STRUCT
display : BOOL; // 显示
setUpDisplay : BOOL; //
number : Int; // 编号
quantity : DInt; // 不良品数量
rate : Real; // 不良率
continuous : DInt; // 连续不良报警数量
cumulative : DInt; // 累计不良报警数量n
cumulativeRange : DInt; // 累计不良计算范围m

END_STRUCT
END_TYPE

// ---- Standard/Public/06 Produce/UDT_BadVar_RD.TcDUT
TYPE UDT_BadVar_RD :
STRUCT
badExecute : BOOL; // 不良触发
goodExecute : Bool; // 良品触发
empty : Bool; // 清空连续不良计数和不良计次列表
continuousAlarm : Bool; // 连续不良报警
cumulativeAlarm : Bool; // 累计不良报警
badRatio : Real; // 不良率
goodIncrements : Int; // 良品增量，每次增加的数量
badIncrements : Int; // 不良增量，每次增加的数量
continuous : DInt; // 当前连续不良计数
num : DInt; // 不良计次
lastIndex : DINT ; // 数组索引
machineNo : UINT; // 不良所属机器号
stationNo : UINT; // 不良所属工站号
badNumList : ARRAY[0..10] OF DINT; // 不良计次列表

END_STRUCT
END_TYPE

// ---- Standard/Public/06 Produce/UDT_ProduceDataRecord_RD.TcDUT
TYPE UDT_ProduceDataRecord_RD :
STRUCT
goodValue : DINT; // 良品数量
badValue : DInt; // 不良品数量
totalValue : DInt; // 总产品数量
cumulativeValue : DInt; // 累计生产数量
yieldRatio : Real; // 良品率
badRatio : Real; // 不良率
 
END_STRUCT
END_TYPE

// ---- Standard/Public/06 Produce/UDT_ProduceData_RD.TcDUT
TYPE UDT_ProduceData_RD :
STRUCT
  goodValue : DINT; // 良品数量
badValue : DInt; // 不良品数量
totalValue : DInt; // 总产品数量
cumulativeValue : DInt; // 累计生产数量
yieldRatio : Real; // 良品率
badRatio : Real; // 不良率

END_STRUCT
END_TYPE

// ---- Standard/Public/06 Produce/UDT_ProduceHmi_RD.TcDUT
TYPE UDT_ProduceHmi_RD :
STRUCT
setUp : BOOL; // 设置中
allClearHmi : Bool; // 全部清零Hmi
percentMode : Int; // 百分比模式  0:  N/总产量, 1:  N/总不良
sortMode : Int; // 排序模式 0:  分类序号, 1:  大->小, 2:  小->大
goodValue : DInt; // 良品数量
badValue : DInt; // 不良品数量
totalValue : DInt; // 总产品数量
cumulativeValue : DInt; // 累计生产数量
badMax : DInt; // 分类不良单项最大数
yieldRatio : Real; // 良品率
badRatio : Real; // 不良率
badMin : DInt; // 分类不良单项最小数
pieChart : ARRAY[0..1] OF Real; // 饼图值
badShow : ARRAY[0..5] OF UDT_BadHmi_RD; // 分类不良显示
turnPages : UDT_TurnPages_RD; // 滚动条

END_STRUCT
END_TYPE

// ---- Standard/Public/06 Produce/UDT_ProduceVar_RD.TcDUT
TYPE UDT_ProduceVar_RD :
STRUCT
goodExecute : BOOL; // 良品计数
allClearHmi : Bool; // 全部清零Hmi
allClearAuto : Bool; // 全部清零Auto
goodIncrements : Int; // 良品增量，每次增加的数量
percentMode : Int; // 百分比模式  0:  N/总产量, 1:  N/总不良
sortMode : Int; // 排序模式 0:  分类序号, 1:  大->小, 2:  小->大
badTypeNum : Int; // 分类不良数量
badMax : DINT; // 分类不良最大值
badList : ARRAY[0..99] OF int; // 下属分类不良编号

END_STRUCT
END_TYPE

// ---- Standard/Public/08 WearPart/UDT_WearPartData_RD.TcDUT
TYPE UDT_WearPartData_RD :
STRUCT
  actUsage : DINT; // 当前使用量
  maxUsage : DInt; // 最大使用量
  tipRate : Real; // 提示比例
  recordsTime : ARRAY[0..9] OF TIMESTRUCT; // 记录时间
  recordsUsage : Array[0..9] of DInt; // 记录用量

END_STRUCT
END_TYPE

// ---- Standard/Public/08 WearPart/UDT_WearPartHmi_RD.TcDUT
TYPE UDT_WearPartHmi_RD :
STRUCT
  actUsage : DINT; // 当前使用量
  maxUsage : DInt; // 最大使用量
  tipRate : Real; // 提示比例
  recordsTime : ARRAY[0..9] OF TIMESTRUCT; // 记录时间
  recordsUsage : ARRAY[0..9] OF DINT; // 记录用量
  clearHmi : BOOL; //清零Hmi
  clearForbidIcon : Bool; //清零禁止图标
END_STRUCT
END_TYPE

// ---- Standard/Public/08 WearPart/UDT_WearPartVar_RD.TcDUT
TYPE UDT_WearPartVar_RD :
STRUCT
countExecute : BOOL; //计数
clearHmi : Bool; //清零Hmi
clearAllow : Bool; //清零允许操作
clearForbidIcon : Bool; //清零禁止图标
clearPermit : Bool; //清零条件
clearAuto : Bool; //清零Auto
display : Bool; //显示
alarming : Bool; //报警
tip : Bool; //提示
machineNo : UINT; //所属机器编号
stationNo : UINT; //所属工站编号
serialNo : UINT; //HMI显示序号
subDisplay : Word; //子页面显示
increments : DInt; //计数增量
unit : ARRAY[0..3] OF STRING[20]; //单位
name : ARRAY[0..3] OF STRING[20]; //名字

END_STRUCT
END_TYPE

// ---- Standard/Public/11 Oee/UDT_OeeData_RD.TcDUT
TYPE UDT_OeeData_RD :
STRUCT
startTimeDisplay          : BOOL; // 开始时刻显示
endTimeDisplay            : BOOL; // 结束时刻显示
goodValue                 : DINT; // 良品数量
badValue                  : DINT; // 不良品数量
totalValue                : DINT; // 总数量
availability              : REAL; // 可用率
performance               : REAL; // 性能指数
quality                   : REAL; // 质量指数
oee                       : REAL; // 综合效率
startTime                 : DATE_AND_TIME; // 开始时刻
endTime                   : DATE_AND_TIME; // 结束时刻
totalTime                 : UDT_DayTime_RD; // 总时间
productiveTime            : UDT_DayTime_RD; // 生产时间
downTime                  : UDT_DayTime_RD; // 计划停机时间
runtime                   : UDT_DayTime_RD; // 运行时间
standbyTime               : UDT_DayTime_RD; // 待机时间
failureTime               : UDT_DayTime_RD; // 故障时间
failureCount              : UINT; // 故障次数

END_STRUCT
END_TYPE

// ---- Standard/Public/11 Oee/UDT_OeeHmi_RD.TcDUT
TYPE UDT_OeeHmi_RD :
STRUCT
start                  : BOOL; // 开始
end                    : BOOL; // 结束
clear                  : BOOL; // 清零
scheduledDown          : BOOL; // 计划停止
startTimeDisplay       : BOOL; // 开始时刻显示
endTimeDisplay         : BOOL; // 结束时刻显示
goodValue              : DINT; // 良品数量
badValue               : DINT; // 不良品数量
totalValue             : DINT; // 总数量
availability           : REAL; // 可用率
performance            : REAL; // 性能指数
quality                : REAL; // 质量指数
oee                    : REAL; // 综合效率
startTime              : ARRAY[0..6] OF INT; // 开始时刻
endTime                : ARRAY[0..6] OF INT; // 结束时刻
totalTime              : UDT_DayTime_RD; // 总时间
productiveTime         : UDT_DayTime_RD; // 生产时间
downTime               : UDT_DayTime_RD; // 计划停机时间
runtime                : UDT_DayTime_RD; // 运行时间
standbyTime            : UDT_DayTime_RD; // 待机时间
failureTime            : UDT_DayTime_RD; // 故障时间
failureCount           : UINT; // 故障次数
number                 : INT; // 编号

END_STRUCT
END_TYPE

// ---- Standard/Public/11 Oee/UDT_OeeVar_RD.TcDUT
TYPE UDT_OeeVar_RD :
STRUCT
start                 : BOOL; // 开始
end                   : BOOL; // 结束
keep                  : BOOL; // 保持
clear                 : BOOL; // 清零
scheduledDown         : BOOL; // 计划停止
running               : BOOL; // 运行中
alarming              : BOOL; // 报警中
goodValue             : DINT; // 良品数量
badValue              : DINT; // 不良数量
idealCycleTime        : TIME; // 理想周期时间
END_STRUCT
END_TYPE

// ---- Standard/Unit/03 Estop/UDT_Estop_RD.TcDUT
TYPE UDT_Estop_RD :
STRUCT
input        : BOOL;
notEstop     : BOOL;
disable      : BOOL;
END_STRUCT
END_TYPE

// ---- Standard/Unit/04 SafetyDoor/UDT_SafetyDoor_RD.TcDUT
TYPE UDT_SafetyDoor_RD :
STRUCT
inputArrived             : BOOL;
inputLocked              : BOOL;
inputUnlockButton        : BOOL;
outputLockCoil           : BOOL;
outputUnlockButtonLight  : BOOL;
notLocked                : BOOL;
prohibitUnlock           : BOOL;
lightWhenLocked          : BOOL;
disabled                 : BOOL;
autoLock                 : BOOL;
autoLockTime             : TIME;
arrivedLabel             : STRING[10];
lockedLabel              : STRING[10];
name                     : ARRAY[0..3] OF STRING[30];
machineNo                : UINT;
END_STRUCT
END_TYPE

// ---- Standard/Unit/05 Cylinder/UDT_CylinderData_RD.TcDUT
TYPE UDT_CylinderData_RD :
STRUCT
homeTime : UDINT; // 原点到位延时
workTime : UDINT; // 动点到位延时
alarmTime : UDINT; // 报警延时
homeSensorDisabled : Array[0..3] of Bool; // 原点传感器屏蔽
workSensorDisabled : Array[0..3] of Bool; // 动点传感器屏蔽
  
END_STRUCT
END_TYPE

// ---- Standard/Unit/05 Cylinder/UDT_CylinderHmi_RD.TcDUT
TYPE UDT_CylinderHmi_RD :
STRUCT 
  
homehmi : BOOL; // 原点hmi
homeForbidIcon : BOOL; // 原点禁止图标
homeValve : BOOL; // 原点阀
homeManual : BOOL; // 原点Manual
workhmi : BOOL; // 动点hmi
workManual : Bool; // 动点Manual
workForbidIcon : Bool; // 动点禁止图标
workValve : BOOL; // 动点阀
homeSensor : ARRAY[0..3] OF BOOL; // 原点传感器
workSensor : Array[0..3] of Bool; // 动点传感器
homeSensorLabel : ARRAY[0..3] OF STRING[10]; // 原点传感器标签
workSensorLabel : Array[0..3] of STRING[10]; // 动点传感器标签
toHomeActionTime : UDINT; // 到原点所用时间
toWorkActionTime : UDINT; // 到动点所用时间

//homeTime : UDINT; // 原点到位延时
//workTime : UDINT; // 动点到位延时



END_STRUCT
END_TYPE

// ---- Standard/Unit/05 Cylinder/UDT_CylinderMessage_RD.TcDUT
TYPE UDT_CylinderMessage_RD :
STRUCT
inManualOperationAutoTip : BOOL; //
noHomePermitManualTip : Bool; //
noWorkPermitManualTip : Bool; //
homeSensorOffAlarm : Array[0..3] of Bool; //
workSensorOffAlarm : Array[0..3] of Bool; //
homeSensorOnAlarm : Array[0..3] of Bool; //
workSensorOnAlarm : Array[0..3] of Bool; //
  
END_STRUCT
END_TYPE

// ---- Standard/Unit/05 Cylinder/UDT_CylinderVar_RD.TcDUT
TYPE UDT_CylinderVar_RD :
STRUCT
homehmi : BOOL; // 原点hmi
homeManual : Bool; // 原点Manual
homeForbidIcon : Bool; // 原点禁止图标
homeValve : Bool; // 原点阀
homeInit : Bool; // 原点Init
homePermit : Bool; // 原点动作条件
noHomePermitManualTip : Bool; // 原点动作条件不满足手动提示
inHome : Bool; // 在原点位
workhmi : Bool; // 动点hmi
workManual : Bool; // 动点Manual
workForbidIcon : Bool; // 动点禁止图标
workValve : Bool; // 动点阀
workInit : Bool; // 动点Init
workPermit : Bool; // 动点动作条件
noWorkPermitManualTip : Bool; // 动点动作条件不满足手动提示
inWork : Bool; // 在动点位
enabled : Bool; // 使能中
release : Bool; // 泄气
busy : Bool; // 运动中
manual : Bool; // 手动执行
auto : Bool; // 自动执行
alarming : Bool; // 报警中
autoTip : Bool; // 自动提示
estoppedReInit : Bool; // 急停后需要重新初始化
display : Bool; // 画面显示
homeSensorOffAlarm : Array[0..3] of Bool; // 原点传感器无信号报警
workSensorOffAlarm : Array[0..3] of Bool; // 动点传感器无信号报警
homeSensorOnAlarm : Array[0..3] of Bool; // 原点传感器有信号报警
workSensorOnAlarm : Array[0..3] of Bool; // 动点传感器有信号报警
homeSensor : Array[0..3] of Bool; // 原点传感器
workSensor : Array[0..3] of Bool; // 动点传感器
homeSensorLabel : Array[0..3] of STRING[10]; // 原点传感器标签
workSensorLabel : Array[0..3] of STRING[10]; // 动点传感器标签
toHomeActionTime : UDINT; // 到原点所用时间
toWorkActionTime : UDINT; // 到动点所用时间
displayCylNum : UINT; // 显示气缸数量
controlCylNum : UINT; // 控制气缸数量
stationNo : UINT; // 所属工站编号
serialNo : UINT; // hmi显示序号
  
END_STRUCT
END_TYPE

// ---- Standard/Unit/06 Axis/UDT_AxisData_RD.TcDUT
TYPE UDT_AxisData_RD :
STRUCT
homeDisplay : BOOL; // 伺服回原点按钮可见
autoVelo : Real; // 自动速度
manualVelo : Real; // 手动速度
jogVelo : REAL; // JOG速度
jogDistance :REAL;//伺服JOG步进量
acceleration : Real; // 加速度
deceleration : Real; // 减速度
movePos : Array[0..31] of Real; // 定位坐标
  
END_STRUCT
END_TYPE

// ---- Standard/Unit/06 Axis/UDT_AxisHmi_RD.TcDUT
TYPE UDT_AxisHmi_RD :
STRUCT
powerhmi : BOOL; // 伺服Onhmi
powerForbidIcon : Bool; // 伺服On禁止图标
isPowerOn : Bool; // 伺服On状态
halthmi : BOOL; // 伺服暂停hmi
resethmi : BOOL;//伺服复位hmi
jogForwardhmi : Bool; // 伺服JOG+_hmi
jogForwardForbidIcon : Bool; // 伺服JOG+禁止图标
jogBackwardshmi : Bool; // 伺服JOG-hmi
jogBackwardsForbidIcon : BOOL; // 伺服JOG-禁止图标
jogDistance :REAL;//伺服JOG步进量
homehmi : Bool; // 伺服回原点hmi
homeForbidIcon : Bool; // 伺服回原点禁止图标
homeDisplay : Bool; // 伺服回原点按钮可见
homeDone : Bool; // 伺服回原点完成
brakehmi : Bool; // 伺服刹车hmi
brakeForbidIcon : Bool; // 伺服刹车禁止图标
brake : Bool; // 伺服刹车输出
movehmi : Bool; // 定位启动hmi
moveForbidIcon : BOOL; // 定位启动禁止图标
movehmiNo : UINT; // 手动定位编号
inPosNo : UINT; // 伺服到位编号
status : UINT; // 伺服状态
driverErrID : DWORD; // 伺服驱动器错误代码
ncErrID :DWORD;// 伺服NC错误代码
warnID : DWORD; // 伺服警告代码
posUnit : STRING[6]; // 位置单位
veloUnit : String[8]; // 速度单位
accDecUnit : WSTRING; // 加/减速度单位
actPos : REAL; // 当前坐标
actVelo : Real; // 当前速度
actTorque : Real; // 当前转矩
targetDistance :REAL;//伺服目标距离
targetVelocity :REAL;//伺服目标速度
posTeach :BOOL;//伺服位置示教

display : Bool; // 画面显示
selectDisplay : Bool; // 位置选择窗口显示
number : INT; // 部件编号
textListNo : Int; // 文本列表编号
movePosNum : Int; // 定位数量
subDisplay : Int; // 子画面显示
selectPageValue : ARRAY[0..8] OF INT; // 位置选择页值
turnPages : UDT_TurnPages_RD; //

autoVelo : Real; // 自动速度
manualVelo : Real; // 手动速度
jogVelo : Real; // JOG速度
acceleration : Real; // 加速度
deceleration : Real; // 减速度
movePos : ARRAY[0..8] OF REAL; // 定位坐标

lsp : BOOL; // 伺服正极限
lsn : Bool; // 伺服负极限
dog : BOOL; // 伺服原点感应



END_STRUCT
END_TYPE

// ---- Standard/Unit/06 Axis/UDT_AxisMessage_RD.TcDUT
TYPE UDT_AxisMessage_RD :
STRUCT
  
notPowerOnAutoTip : BOOL; // 伺服未On自动提示
error : Bool; // 伺服错误中
notPowerOnManualTip : Bool; // 未使能不能操作
unableBrakeManualTip : Bool; // 已使能不能操作刹车
unablePowerOnManualTip : Bool; // 刹车已打开不能操作使能
notMovePermitManualTip : Int; // 定位条件不满足手动提示
notInPosAutoTip : Int; // 伺服不在位自动提示
  
END_STRUCT
END_TYPE

// ---- Standard/Unit/06 Axis/UDT_AxisVar_RD.TcDUT
TYPE UDT_AxisVar_RD :
STRUCT
powerhmi : BOOL; // 伺服Onhmi
powerManual : Bool; // 伺服OnManual
powerAuto : Bool; // 伺服OnAuto
powerInit : Bool; // 伺服OnInit
powerAllow : Bool; // 伺服On允许操作
powerForbidIcon : Bool; // 伺服On禁止图标
isPowerOn : Bool; // 伺服On状态
notPowerOnAutoTip : Bool; // 伺服未On自动提示
halthmi : BOOL; // 伺服暂停hmi
resethmi : BOOL;//伺服复位hmi
haltManual : Bool; // 伺服暂停Manual
haltAuto : Bool; // 伺服暂停Auto
jogForwardhmi : Bool; // 伺服JOG+_hmi
jogForwardAllow : Bool; // 伺服JOG+允许操作
jogForwardForbidIcon : Bool; // 伺服JOG+禁止图标
jogForwardAuto : Bool; // 伺服JOG+_Auto
jogForwardPermit : Bool; // 伺服JOG+_条件
jogBackwardshmi : Bool; // 伺服JOG-hmi
jogBackwardsAllow : Bool; // 伺服JOG-允许操作
jogBackwardsForbidIcon : Bool; // 伺服JOG-禁止图标
jogBackwardsAuto : Bool; // 伺服JOG-Auto
jogBackwardsPermit : BOOL; // 伺服JOG-条件
homehmi : BOOL; // 伺服回原点hmi
homeManual : Bool; // 伺服回原点Manual
homeAllow : Bool; // 伺服回原点允许操作
homeForbidIcon : Bool; // 伺服回原点禁止图标
homeDisplay : Bool; // 伺服回原点按钮可见
homeDone : Bool; // 伺服回原点完成
homeInit : Bool; // 伺服回原点Init
homing : Bool; // 伺服回原点中
homePermit : Bool; // 伺服回原点条件
notHomeAutoTip : Bool; // 伺服未回原点自动提示
brakeEnable : Bool; // 伺服刹车启用
brakehmi : Bool; // 伺服刹车hmi
brakeAllow : Bool; // 伺服刹车允许操作
brakeForbidIcon : Bool; // 伺服刹车禁止图标
brakeManual : Bool; // 伺服刹车Manual
brake : Bool; // 伺服刹车输出
brakeForced : Bool; // 伺服刹车强制打开输出
movehmi : Bool; // 定位启动hmi
moveAllow : Bool; // 定位启动允许操作
moveForbidIcon : Bool; // 定位启动禁止图标
ready : Bool; // 伺服准备就绪
busy : Bool; // 伺服忙
error : Bool; // 伺服错误
alarming : Bool; // 伺服报警中
warning : Bool; // 伺服警告
timeout : Bool; // 定位超时报警
manualTip : Bool; // 手动提示
autoTip : Bool; // 自动提示
movePermit : Bool; // 定位总条件
eStoppedReInit : Bool; // 急停时是否需要重新初始化
lsp : Bool; // 伺服正极限
lsn : Bool; // 伺服负极限
dog : Bool; // 伺服原点感应
display : Bool; // 画面显示
autoReturning : Bool; // 自动回位中
autoReturnAllow : Bool; // 自动回位已激活待启动
autoReturnPermit : Bool; // 自动回位条件(大范围回位)
autoReturnEnable : Bool; // 自动回位启用
notPowerOnManualTip : Bool; // 未使能不能操作
unableBrakeManualTip : Bool; // 已使能不能操作刹车
unablePowerOnManualTip : Bool; // 刹车已打开不能操作使能
autoReturnScope : Real; // 自动回位范围，在范围内不判断定位条件
homeMode : UINT; // 回原点模式
brakeState : UINT; // 伺服刹车状态
inPosTime : Time; // 到位延时
inPosScope : Real; // 到位范围
actPos : Real; // 当前坐标
actVelo : Real; // 当前速度
actTorque : Real; // 当前转矩
differentVelo : Real; // 自定义速度
driverErrID : DWORD; // 伺服驱动器错误代码
ncErrID :DWORD;// 伺服NC错误代码
warnID : DWord; // 伺服警告代码
modulo : UDT_ModuloProperty_RD; // 模长轴控制
notMovePermitManualTip : UINT; // 定位条件不满足手动提示
notInPosAutoTip : UINT; // 伺服不在位自动提示
movehmiNo : UINT; // 手动定位编号
moveAutoNo : UINT; // 自动定位编号
moveAutoNoCache : UINT; // 自动定位编号暂存
status : UINT; // 伺服状态
movePosNum : UINT; // 定位数量
stationNo : UINT; // 工站编号
serialNo : UINT; // 在工站内的序号
subDisplay : Word; // 子画面显示
axis : AXIS_REF; // 轴引用
posUnit : String[6]; // 位置单位
veloUnit : String[8]; // 速度单位
accDecUnit : WSTRING; // 加/减速度单位
name : Array[0..3] of String[30]; // 伺服名称
absOrRel : Array[0..31] of Bool; // 绝对/相对定位
inPos : Array[0..31] of Bool; // 定位到位
movePermits : ARRAY[0..31] OF BOOL; // 定位条件


velocityHmi     : BOOL; // 伺服速度模式hmi
velocityAuto    : BOOL; // 伺服速度模式Auto
VelocityAllow   : BOOL; // 伺服速度允许操作
VelocityPermit   : BOOL; // 伺服速度动作条件
velocityBusy		: BOOL;	//伺服速度模式Busy
velocityError		: BOOL;	//伺服速度模式Error
velocityErrorID	: UDINT;	//伺服速度模式ErrorID
inVelocity	    : BOOL;	 //速度到达
velocity		    : REAL;	//轴速度模式速度
 
stophmi : BOOL; // 伺服停止hmi
stopManual : BOOL; // 伺服停止Manual
stopAuto : BOOL; // 伺服停止Auto

additiveAuto : BOOL;
additiveDistance : REAL;
additiveVelo : REAL;

inPosNo : UINT; // 伺服到位编号
targetDistance :REAL;//伺服目标距离
targetVelocity :REAL;//伺服目标速度
posTeach :BOOL;//伺服位置示教
Override : INT; // 速度百分比

 
END_STRUCT
END_TYPE

// ---- Standard/Unit/06 Axis/UDT_ModuloProperty_RD.TcDUT
TYPE UDT_ModuloProperty_RD :
STRUCT
enable : BOOL; //启用模长
inCalibratePos : Bool; //在标定位置
inClosestPos : Bool; //在分割点位置
inAutoPos : Bool; //在自动分割点位置
inAutoNextPos : Bool; //在自动下一个分割点位置
calibrateOffset : Real; //标定位置与分割点偏移值
tolerance : Real; //公差范围
factor : Real; //模长
mode : Int; //模式，0:分度盘模式 1:棘轮模式
divisor : Int; //分割数
stepPoint : Int; //单次进给/后退量  MAX<Divisor
actPoint : Int; //当前分割点
closestPoint : Int; //当前最近分割点
previousPoint : Int; //当前上一分割点
nextPoint : Int; //当前下一分割点
autoNextPoint : Int; //自动下一分割点
autoPoint : Int; //自动应该在割点
closestPos : Real; //当前最近分割点坐标
previousPos : Real; //当前上一分割点坐标
nextPos : Real; //当前下一分割点坐标
autoPos : Real; //自动应该在分割点坐标
autoNextPos : Real; //自动下一分割点坐标
moveMode : ARRAY[0..6] OF INT; //定位模式

  
END_STRUCT
END_TYPE

// ---- Standard/Unit/07 Sensor/UDT_SensorData_RD.TcDUT
TYPE UDT_SensorData_RD :
STRUCT
disabled         : BOOL; //传感器屏蔽
setCount         : UINT; //传感器异常报警次数设置
onTime           : UDINT; //On延时时间值
offTime          : UDINT; //Off延时时间值
flickerTime      : UDINT; //闪烁延时时间值

END_STRUCT
END_TYPE

// ---- Standard/Unit/07 Sensor/UDT_SensorHmi_RD.TcDUT
TYPE UDT_SensorHmi_RD :
STRUCT
subDisplay : BOOL; //子画面显示
input : Bool; //传感器输入
display : Bool; //画面显示
count : Int; //感应器异常计次
label : String[10]; //传感器标签
disabled : Bool; //传感器屏蔽
setCount : Int; //传感器异常报警次数设置
onTime : DINT; //On延时时间值
offTime : DINT; //Off延时时间值
flickerTime : DINT; //闪烁延时时间值
number : INT; //部件编号
  
END_STRUCT
END_TYPE

// ---- Standard/Unit/07 Sensor/UDT_SensorVar_RD.TcDUT
TYPE UDT_SensorVar_RD :
STRUCT
input            : BOOL; // 传感器输入
check            : BOOL; // 传感器异常检测,On开始 Off结束，外部触发
isOn             : BOOL; // On延时输出
isOff            : BOOL; // Off延时输出
unchangeError    : BOOL; // 输入信号状态无变化异常报警
flickerError     : BOOL; // 输入信号频繁闪烁异常报警
alarming         : BOOL; // 报警中
display          : BOOL; // 显示
subDisplay       : BOOL; // 子画面显示
count            : UINT; // 感应器异常计次
stationNo        : UINT; // 所属工站编号
serialNo         : UINT; // 在工站内的序号
label            : STRING[10]; // 传感器标签
END_STRUCT
END_TYPE

// ---- Standard/Unit/08 Motor/UDT_MotorData_RD.TcDUT
TYPE UDT_MotorData_RD :
STRUCT
startTime       : DINT;// 启动延时
stopTime        : DINT;// 停止延时
END_STRUCT
END_TYPE

// ---- Standard/Unit/08 Motor/UDT_MotorHmi_RD.TcDUT
TYPE UDT_MotorHmi_RD :
STRUCT
inputRunning          : BOOL;//运行监控输入
inputError            : BOOL;// 错误输入
outputForward         : BOOL;// 正转输出
outputReversal        : BOOL;// 反转输出
outputErrorReset      : BOOL;// 错误复位输出
forwardHmi            : BOOL;// 正转HMI
forwardForbidIcon     : BOOL;// 正转禁止图标
reversalHmi           : BOOL;// 反转HMI
reversalForbidIcon    : BOOL;// 反转禁止图标
display               : BOOL;// 显示
forwardHmiState       : INT;// 正转Hmi状态
reversalHmiState      : INT;// 反转Hmi状态
number                : INT;// 编号
startTime             : DINT;// 启动延时
stopTime              : DINT;// 停止延时
END_STRUCT
END_TYPE

// ---- Standard/Unit/08 Motor/UDT_MotorVar_RD.TcDUT
TYPE UDT_MotorVar_RD :
STRUCT
inputRunning        : BOOL;// 运行监控输入
inputError          : BOOL;// 错误输入
outputForward       : BOOL;// 正转输出
outputReversal      : BOOL;// 反转输出
outputErrorReset    : BOOL;// 错误复位输出
forwardHmi          : BOOL;// 正转HMI
forwardForbidIcon   : BOOL;// 正转禁止图标
forwardManual       : BOOL;// 正转手动执行
forwardAuto         : BOOL;// 正转自动执行
forwardManualTip    : BOOL;// 正转手动提示
forwardPermit       : BOOL;// 正转条件
inForward           : BOOL;// 正转运行中
reversalHmi         : BOOL;// 反转HMI
reversalForbidIcon  : BOOL;// 反转禁止图标
reversalManual      : BOOL;// 反转手动执行
reversalAuto        : BOOL;// 反转自动执行
reversalManualTip   : BOOL;// 反转手动提示
reversalPermit      : BOOL;// 反转条件
inReversal          : BOOL;// 反转运行中
init                : BOOL;// 初始化
alarming            : BOOL;// 报警中
autoTip             : BOOL;// 自动提示中
runningAlarm        : BOOL;// 运行监控报警
inverterAlarm       : BOOL;// 变频器报警
forwardHmiState     : UINT;// 正转Hmi状态
reversalHmiState    : UINT;// 反转Hmi状态
monitorMode         : UINT;// 监控模式: 0停用运行监控 1启用运行监控
turnMode            : UINT;// 运转模式: 1正转 2反转 3正反转
stationNo           : UINT;// 所属工站编号
serialNo            : UINT;// HMI显示序号
END_STRUCT
END_TYPE

// ---- Standard/Unit/11 KeyenceScan/UDT_KeyenceScanData_RD.TcDUT
TYPE UDT_KeyenceScanData_RD :
STRUCT
evaluationGrade     : UINT; // 评价等级下限 4:A  3:B  2:C  1:D  0:F
evaluationMode      : UINT; // 评价等级方式 0:不评估  1:ISO/IEC15415  2:ISO/IEC TR 29158
timeout             : TIME; // 超时设置
END_STRUCT
END_TYPE

// ---- Standard/Unit/11 KeyenceScan/UDT_KeyenceScanHmi_RD.TcDUT
TYPE UDT_KeyenceScanHmi_RD :
STRUCT
triggerHmi           : BOOL; // 触发Hmi
triggerManual        : BOOL; // 触发Manual
triggerForbidIcon    : BOOL; // 触发禁止图标
ready                : BOOL; // 准备就绪
busy                 : BOOL; // 流程控制中
done                 : BOOL; // 完成
display              : BOOL; // 显示
disabled             : BOOL; // 屏蔽
alarming             : BOOL; // 报警中
subDisplay           : WORD; // 子页面显示
resultData           : STRING[128]; // 扫码结果数据
readResultCode       : INT; // 读取动作错误代码
generalErrorCode     : INT; // 一般错误代码
scanGrade            : INT; // 扫码等级
result               : INT; // 结果寄存器 1:Pass  2:Fail 3:Timeout
status               : UINT; //7
sensorSeries         : STRING[10]; // 传感器系列, 范围：N-L20,SR-1000X,SR-2000X,SR-LR1
number               : INT; //编号
evaluationGrade      : INT; // 评价等级下限 4:A  3:B  2:C  1:D  0:F
evaluationMode       : INT; // 评价等级方式 0:不评估  1:ISO/IEC15415  2:ISO/IEC TR 29158
timeout              : DINT; // 超时设置
END_STRUCT 
END_TYPE

// ---- Standard/Unit/11 KeyenceScan/UDT_KeyenceScanVar_RD.TcDUT
TYPE UDT_KeyenceScanVar_RD :
STRUCT
triggerHmi          : BOOL; // 触发Hmi
triggerManual       : BOOL; // 触发Manual
triggerAuto         : BOOL; // 触发Auto
triggerAllow        : BOOL; // 触发允许操作
triggerForbidIcon   : BOOL; // 触发禁止图标
ready               : BOOL; // 准备就绪
busy                : BOOL; // 流程控制中
done                : BOOL; // 完成
disabled            : BOOL; // 屏蔽
alarming            : BOOL; // 报警中
readTimeoutDisabled : BOOL; // 读取超时报警屏蔽
subDisplay          : WORD; // 子页面显示
readTimeoutAlarm    : BOOL; // 超时报警
readError           : BOOL; // 读取动作错误
generalError        : BOOL; // 一般错误
resultData          : STRING[128]; // 扫码结果数据
readResultCode      : UINT; // 读取动作错误代码
generalErrorCode    : UINT; // 一般错误代码
scanGrade           : UINT; // 扫码等级
result              : UINT; // 结果寄存器 1:Pass  2:Fail 3:Timeout
status              : UINT; // 状态
sensorSeries        : STRING[10]; // 传感器系列, 范围：N-L20,SR-1000X,SR-2000X,SR-LR1
stationNo           : UINT; // 所属工站编号
serialNo            : UINT; // HMI显示序号
input               : ARRAY[0..85] OF WORD; // 输入字
output              : ARRAY[0..37] OF WORD; // 输出字

END_STRUCT
END_TYPE

// ---- Standard/Unit/12 Delay/UDT_DelayData_RD.TcDUT
TYPE UDT_DelayData_RD :
STRUCT
setTime               : TIME; // 延时Data
END_STRUCT
END_TYPE

// ---- Standard/Unit/12 Delay/UDT_DelayHmi_RD.TcDUT
TYPE UDT_DelayHmi_RD :
STRUCT
isOn                 : BOOL; // On延时输出
display              : BOOL; // 显示
actTime              : DINT; // 当前计时时间
setTime              : DINT; // 设置延时时间值
number               : INT; // 编号
END_STRUCT
END_TYPE

// ---- Standard/Unit/12 Delay/UDT_DelayVar_RD.TcDUT
TYPE UDT_DelayVar_RD :
STRUCT
input               : BOOL; // 延时开始
isOn                : BOOL; // On延时输出
actTime             : TIME; // 当前计时时间
stationNo           : UINT; // 所属工站编号
serialNo            : UINT; // HMI显示序号
END_STRUCT
END_TYPE

// ---- Standard/Unit/13 Valve/UDT_ValveData_RD.TcDUT
TYPE UDT_ValveData_RD :
STRUCT
holdTime       : TIME; // 阀动作保持时间
END_STRUCT
END_TYPE

// ---- Standard/Unit/13 Valve/UDT_ValveHmi_RD.TcDUT
TYPE UDT_ValveHmi_RD :
STRUCT
hmi           : BOOL; // HMI
manual        : BOOL; // 手动执行
forbidIcon    : BOOL; // 禁止图标
display       : BOOL; // 显示
valve         : BOOL; // 阀输出
number        : INT; // 编号
holdTime      : DINT; // 阀动作保持时间
END_STRUCT 
END_TYPE

// ---- Standard/Unit/13 Valve/UDT_ValveVar_RD.TcDUT
TYPE UDT_ValveVar_RD :
STRUCT
hmi        : BOOL; // HMI
manual     : BOOL; // 手动执行
allow      : BOOL; // 允许操作
forbidIcon : BOOL; // 禁止图标
permit     : BOOL; // 动作条件
auto       : BOOL; // 自动执行
init       : BOOL; // 初始化执行
manualTip  : BOOL; // 手动提示
autoTip    : BOOL; // 自动提示
isOn       : BOOL; // 延时到位
valve      : BOOL; // 阀输出
stationNo  : UINT; // 所属工站编号
serialNo   : UINT; // HMI显示序号
END_STRUCT
END_TYPE

// ---- Standard/Unit/40 RackFeeder/UDT_RackFeederData_RD.TcDUT
TYPE UDT_RackFeederData_RD :
STRUCT
  
rollLimit : INT; // 卷纸马达10秒内转圈数上限
startTime : Time; // 启动延时
stopTime : Time; // 停止延时
timeout : Time; // 放料超时延时

END_STRUCT
END_TYPE

// ---- Standard/Unit/40 RackFeeder/UDT_RackFeederHmi_RD.TcDUT
TYPE UDT_RackFeederHmi_RD :
STRUCT
input : UDT_RackFeederInput_RD; //
output : UDT_RackFeederOutput_RD; //
ready : BOOL; // 准备就绪
alarming : BOOL; // 报警中
feedHmi : BOOL; // 放料马达HMI
feedManual : BOOL; // 放料马达Manual
feedForbidIcon : BOOL; // 放料马达禁止图标
rollHmi : BOOL; // 卷纸马达HMI
rollManual : BOOL; // 卷纸马达Manual
rollForbidIcon : BOOL; // 卷纸马达禁止图标
display : BOOL; // 显示
tail : BOOL; // 尾料模式，缺料时不提示
breakLabel : String[10]; // 纸带断裂检测标签
scatterLabel : String[10]; // 散料检测标签
fullLabel : String[10]; // 满料检测标签
number : Int; //编号
rollLimit : Int; // 卷纸马达10秒内转圈数上限
startTime : UDINT; // 启动延时
stopTime : UDINT; // 停止延时
timeout : UDINT; // 放料超时延时

END_STRUCT
END_TYPE

// ---- Standard/Unit/40 RackFeeder/UDT_RackFeederInput_RD.TcDUT
TYPE UDT_RackFeederInput_RD :
STRUCT
full : BOOL; // 满料检测
break : BOOL; // 纸带断裂检测
scatter : BOOL; // 散料检测
feedButton : BOOL; // 放料按钮

END_STRUCT
END_TYPE

// ---- Standard/Unit/40 RackFeeder/UDT_RackFeederOutput_RD.TcDUT
TYPE UDT_RackFeederOutput_RD :
STRUCT
  
feedStart : BOOL; // 放料马达启动
rollStart : BOOL; // 卷纸马达启动

END_STRUCT
END_TYPE

// ---- Standard/Unit/40 RackFeeder/UDT_RackFeederVar_RD.TcDUT
TYPE UDT_RackFeederVar_RD :
STRUCT
input : UDT_RackFeederInput_RD; //
output : UDT_RackFeederOutput_RD; //
ready : BOOL; // 准备就绪
alarming : BOOL; // 报警中
manualTip : BOOL; // 手动提示
tip : BOOL; // 一般提示
feedHmi : BOOL; // 放料马达HMI
feedManual : BOOL; // 放料马达Manual
feedAllow : BOOL; // 放料马达允许操作
feedForbidIcon : BOOL; // 放料马达禁止图标
rollHmi : BOOL; // 卷纸马达HMI
rollManual : BOOL; // 卷纸马达Manual
rollAllow : BOOL; // 卷纸马达允许操作
rollForbidIcon : BOOL; // 卷纸马达禁止图标
display : BOOL; // 显示
disabled : BOOL; // 不启用，料号配方里未用到该部品
tail : BOOL; // 尾料模式，缺料时不提示
timeoutAlarm : BOOL; // 放料超时报警
breakAlarm : BOOL; // 纸带断裂报警
scatterAlarm : BOOL; // 散料报警
stationNo : Int; // 所属工站编号
serialNo : Int; // HMI显示序号
breakLabel : String[10]; // 纸带断裂检测标签
scatterLabel : String[10]; // 散料检测标签
fullLabel : String[10]; // 满料检测标签


END_STRUCT
END_TYPE

// ---- Standard/Unit/40 RackFeeder/UDT_RackFeedMessage_RD.TcDUT
TYPE UDT_RackFeedMessage_RD :
STRUCT
tail : BOOL; // 尾料模式，缺料时不提示
timeoutAlarm : BOOL; // 放料超时报警
breakAlarm : BOOL; // 纸带断裂报警
scatterAlarm : BOOL; // 散料报警

END_STRUCT
END_TYPE

// ---- GVLs/GVL_Module.TcGVL
VAR_GLOBAL
 {attribute 'OPC.UA.DA' := '1'}
  JS : UDT_JacketStripping_RD;
 {attribute 'OPC.UA.DA' := '1'}  
  BF : UDT_BraidFlaring_RD;
{attribute 'OPC.UA.DA' := '1'}  
  CP : UDT_Crimping_RD;
END_VAR

VAR_GLOBAL PERSISTENT
  {attribute 'OPC.UA.DA' := '1'}
  JSData : UDT_Data_JacketStripping_RD;
  {attribute 'OPC.UA.DA' := '1'}  
  BFData : UDT_Data_BraidFlaring_RD;
  {attribute 'OPC.UA.DA' := '1'}  
  CPData : UDT_Data_Crimping_RD;
END_VAR

// ---- GVLs/GVL_Constant.TcGVL
VAR_GLOBAL CONSTANT



BOWL_FEEDER_NUM : UINT :=3; //振动盘数量,范围:0 - 30
BAD_TYPE_NUM : UINT :=10; //不良品类型数量,范围:0 - 30

RFID_NUM : UINT :=2; //RFID数量,范围:0 - 30
WEAR_PART_NUM : UINT :=10; //易损件数量,范围:0 - 30
CCD_NUM : UINT :=2; //CCD数量,范围:0 - 30


CKD_NUM : UINT :=2; //CKD转台数量,范围:0 - 10
vacuum_NUM : UINT :=2; //真空发生器数量,范围:0 - 300


PART_NO_NUM : UINT :=30; //多料号数量,范围:1 - 100
KEYENCE_IV_NUM : UINT :=2; //KEYENCE IV系列传感器数量,范围:0 - 30
WEISS_NUM : UINT :=2; //Weiss转台数量,范围:0 - 10
KEYENCE_MARKING_NUM : UINT :=2; //KEYENCE MD-X系列激光打码数量,范围:0 - 30
KEYENCE_IX_NUM : UINT :=2; //KEYENCE IX系列传感器数量,范围:0 - 30
KEYENCE_GT_NUM : UINT :=2; //KEYENCE GT2、GT、IL、IG的高度传感器数量,范围:0 - 30
RACK_FEEDER_NUM : UINT :=5; //料架数量,范围:0 - 30
FEEDING_NUM : UINT :=10; //进料数量,范围:0 - 30
AXIS_POS_NUM : UINT :=24; //单轴定位数量,范围:8 - 64
DATALOGIC_SCAN_NUM : UINT :=2; //Datalogic DM系列扫码枪数量,范围:0 - 30
HONEYWELL_SCAN_NUM : UINT :=10; //Honeywell扫码枪数量,范围:0 - 30
RCON_NUM : UINT :=2; //IAI电缸数量,范围:0 - 30
EPSON_ROBOT_NUM : UINT :=2; //EPSON机器人数量,范围:0 - 4


MACHINE_NUM : UINT :=1; //机器数量,范围:1 - 4
STATION_NUM : UINT :=20; //工站数量,范围:1 - 50
CYLINDER_NUM : UINT :=100; //气缸数量,范围:0 - 300
AXIS_NUM : UINT :=12; //TO轴数量,范围:0 - 30
ESTOP_NUM : UINT :=10; //急停数量,范围:0 - 100
SAFETY_DOOR_NUM : UINT :=10; //安全门数量,范围:0 - 100
SENSOR_NUM : UINT :=50; //检测传感器数量,范围:0 - 300
DELAY_NUM : UINT :=50; //延时数量,范围:0 - 300
MOTOR_NUM : UINT :=5; //普通马达数量,范围:0 - 100
PRODUCE_NUM: UINT :=1;
OEE_NUM: UINT :=1;
KEYENCE_SCAN_NUM : UINT :=2; //KEYENCE SR系列扫码枪数量,范围:0 - 30
VALVE_NUM : UINT :=20; //单阀数量,范围:0 - 300


HMI_NUM : UINT :=2; //HMI数量,范围:1 - 6



SMC_IONIZER_NUM : UINT :=2; //SMC离子发生器数量,范围:0 - 100
DUMMY_NUM : UINT :=10; //点检数量,范围:0 - 50
SMC_ELECTRIC_CYL_NUM : UINT :=2; //SMC电缸数量,范围:0 - 30
AXIS_EPOS_NUM : UINT :=2; //EPOS轴数量,范围:0 - 30
ATEQ_NUM : UINT :=2; //ATEQ泄露仪数量,范围:0 - 30
COSMO_NUM : UINT :=2; //COSMO泄露仪数量,范围:0 - 30
COGNEX_CAMERA_NUM : UINT :=1; //Cognex In-Sight相机数量,范围:0 - 30
COGNEX_SCAN_NUM : UINT :=1; //Cognex DataMan系列扫码枪数量,范围:0 - 30
KEYENCE_CAMERA_NUM : UINT :=5; //KEYENCE CV-X、XG-X系列相机数量,范围:0 - 30
OMRON_CAMERA_NUM : UINT :=2; //Omron FH系列相机数量,范围:0 - 30

TEST  : UINT :=0;

END_VAR

// ---- GVLs/GVL_Standard.TcGVL
VAR_GLOBAL

Machine : ARRAY[1..MACHINE_NUM] OF UDT_Machine_RD; 
Station : ARRAY[1..STATION_NUM] OF UDT_Station_RD;
CylinderVar : ARRAY[0..CYLINDER_NUM] OF UDT_CylinderVar_RD;
CylinderData : ARRAY[0..CYLINDER_NUM] OF UDT_CylinderData_RD;
AxisVar : ARRAY[0..AXIS_NUM] OF UDT_AxisVar_RD; 
AxisData : ARRAY[0..AXIS_NUM] OF UDT_AxisData_RD; 
Estop : ARRAY[0..ESTOP_NUM] OF UDT_Estop_RD; //
SafetyDoor : ARRAY[0..SAFETY_DOOR_NUM] OF UDT_SafetyDoor_RD; //
SensorVar : ARRAY[0..SENSOR_NUM] OF UDT_SensorVar_RD; //
SensorData : ARRAY[0..SENSOR_NUM] OF UDT_SensorData_RD; //
DelayVar : ARRAY[0..DELAY_NUM] OF UDT_DelayVar_RD; //
DelayData : ARRAY[0..DELAY_NUM] OF UDT_DelayData_RD; //
MotorVar : ARRAY[0..MOTOR_NUM] OF UDT_MotorVar_RD; //
MotorData : ARRAY[0..MOTOR_NUM] OF UDT_MotorData_RD; //
ValveVar : ARRAY[0..VALVE_NUM] OF UDT_ValveVar_RD; //
ValveData : ARRAY[0..VALVE_NUM] OF UDT_ValveData_RD; //


ProduceVar : ARRAY[0..PRODUCE_NUM] OF UDT_produceVar_RD; 
ProduceData : ARRAY[0..PRODUCE_NUM] OF UDT_produceData_RD; 
ProduceDataRecord : ARRAY[0..PRODUCE_NUM] OF UDT_ProduceDataRecord_RD;
badVar : ARRAY[0..BAD_TYPE_NUM] OF UDT_badVar_RD; 
badData : ARRAY[0..BAD_TYPE_NUM] OF UDT_badData_RD; 
WearPartVar : ARRAY[0..WEAR_PART_NUM] OF UDT_WearPartVar_RD; //
WearPartData : ARRAY[0..WEAR_PART_NUM] OF UDT_WearPartData_RD; //

OeeVar : ARRAY[0..OEE_NUM] OF UDT_OeeVar_RD; 
OeeData : ARRAY[0..OEE_NUM] OF UDT_OeeData_RD; 
OeeLastData : ARRAY[0..OEE_NUM] OF UDT_OeeData_RD;

Hmi : ARRAY[1..HMI_NUM] OF UDT_Hmi_RD;

System : UDT_System_RD;
KeyenceScanVar : ARRAY[0..OEE_NUM] OF UDT_KeyenceScanVar_RD; 
KeyenceScanData : ARRAY[0..OEE_NUM] OF UDT_KeyenceScanData_RD; 

  
END_VAR

VAR_GLOBAL
  
fbMachine : ARRAY[1..MACHINE_NUM] OF FB_Machine_RD; //
fbstation : ARRAY[1..STATION_NUM] OF FB_Station_RD; //
fbCylinder : ARRAY[0..CYLINDER_NUM] OF FB_Cylinder_RD; //
fbAxis : ARRAY[0..AXIS_NUM] OF FB_Axis_RD; 
fbEstop : ARRAY[0..ESTOP_NUM] OF FB_Estop_RD; //
fbSafetyDoor : ARRAY[0..SAFETY_DOOR_NUM] OF FB_SafetyDoor_RD; //
fbSensor : ARRAY[0..SENSOR_NUM] OF FB_Sensor_RD; //
fbDelay : ARRAY[0..DELAY_NUM] OF FB_Delay_RD; //
fbMotor : ARRAY[0..MOTOR_NUM] OF FB_Motor_RD; //

fbProduce : ARRAY[1..PRODUCE_NUM] OF FB_Produce; //
fbWearPart : ARRAY[1..WEAR_PART_NUM] OF FB_WearPart;//

fbOee : ARRAY[1..OEE_NUM] OF FB_Oee_RD; //
fbKeyenceScan : ARRAY[0..10] OF FB_KeyenceScan_RD; //
fbTerminal : ARRAY[0..10] OF FB_Terminal_RD; //
fbRackFeeder : ARRAY[0..10] OF FB_RackFeeder_RD; //
fbValve : ARRAY[0..10] OF FB_Valve_RD; //

fbGetPlcClock : FB_GetPlcClock; 

END_VAR

// ---- POUs/MAIN.TcPOU
PROGRAM MAIN
VAR

END_VAR

CallStandardModule();
CallStandard();

END_PROGRAM

// ---- Standard/CallStandardModule.TcPOU
PROGRAM CallStandardModule
VAR
  fbTest  : FB_JacketStripping_RD;
  fbtest2 : FB_BraidFlaring_RD;
  fbtest3 : FB_Crimping_RD; 
  
END_VAR

fbTest(
	JacketStripping:= JS, 
	JacketStrippingData:= JSData, 
  
	homeValve_blow:= , 
	workValve_blow:= , 
  
	homeSensor_gripCyl:= , 
	workSensor_gripCyl:= , 
	homeValve_gripCyl:= , 
	workValve_gripCyl:= , 
	homeLabel_gripCyl:= 'I010100', 
	workLabel_gripCyl:= 'I010101', 
  
	homeSensor_jackCyl:= , 
	workSensor_jackCyl:= , 
	homeValve_jackCyl:= , 
	workValve_jackCyl:= , 
	homeLabel_jackCyl:= 'I010102', 
	workLabel_jackCyl:= 'I010103', 
  
	homeSensor_fixCyl:= , 
	workSensor_fixCyl:= , 
	homeValve_fixCyl:= , 
	workValve_fixCyl:= , 
	homeLabel_fixCyl:= 'I010104', 
	workLabel_fixCyl:= 'I010105', 
  
	homeSensor_stepFixCyl:= , 
	workSensor_stepFixCyl:= , 
	homeValve_stepFixCyl:= , 
	workValve_stepFixCyl:= , 
	homeLabel_stepFixCyl:= 'I010106', 
	workLabel_stepFixCyl:= 'I010107');

  fbtest2(
	BraidFlaring:= BF, 
	BraidFlaringData:= BFData, 
	HomeSensor_gripCyl:= , 
	WorkSensor_gripCyl:= , 
	HomeValve_gripCyl:= , 
	WorkValve_gripCyl:= , 
	HomeLabel_gripCyl:= , 
	WorkLabel_gripCyl:= , 
	HomeSensor_jackCyl:= , 
	WorkSensor_jackCyl:= , 
	HomeValve_jackCyl:= , 
	WorkValve_jackCyl:= , 
	HomeLabel_jackCyl:= , 
	WorkLabel_jackCyl:= , 
	HomeSensor_pushCyl:= , 
	WorkSensor_pushCyl:= , 
	HomeValve_pushCyl:= , 
	WorkValve_pushCyl:= , 
	HomeLabel_pushCyl:= , 
	WorkLabel_pushCyl:= , 
	HomeValve_blow:= , 
	WorkValve_blow:= , 
	HomeValve_vacuum:= , 
	WorkValve_vacuum:= , 
	pushRodInPos:= , 
	HomeSensor_fixCyl:= , 
	WorkSensor_fixCyl:= , 
	HomeValve_fixCyl:= , 
	WorkValve_fixCyl:= , 
	HomeLabel_fixCyl:= , 
	WorkLabel_fixCyl:= , 
	HomeSensor_stepFixCyl:= , 
	WorkSensor_stepFixCyl:= , 
	HomeValve_stepFixCyl:= , 
	WorkValve_stepFixCyl:= , 
	HomeLabel_stepFixCyl:= , 
	WorkLabel_stepFixCyl:= );
	
fbtest3(
	Crimping:= CP, 
	CrimpingData:= CPData, 
	HomeSensor_gripCyl:= , 
	WorkSensor_gripCyl:= , 
	HomeValve_gripCyl:= , 
	WorkValve_gripCyl:= , 
	HomeLabel_gripCyl:= , 
	WorkLabel_gripCyl:= , 
	HomeSensor_jack1Cyl:= , 
	WorkSensor_jack1Cyl:= , 
	HomeValve_jack1Cyl:= , 
	WorkValve_jack1Cyl:= , 
	HomeLabel_jack1Cyl:= , 
	WorkLabel_jack1Cyl:= , 
	HomeSensor_jack2Cyl:= , 
	WorkSensor_jack2Cyl:= , 
	HomeValve_jack2Cyl:= , 
	WorkValve_jack2Cyl:= , 
	HomeLabel_jack2Cyl:= , 
	WorkLabel_jack2Cyl:= , 
	HomeSensor_cutCyl:= , 
	WorkSensor_cutCyl:= , 
	HomeValve_cutCyl:= , 
	WorkValve_cutCyl:= , 
	HomeLabel_cutCyl:= , 
	WorkLabel_cutCyl:= , 
	HomeSensor_feedCyl:= , 
	WorkSensor_feedCyl:= , 
	HomeValve_feedCyl:= , 
	WorkValve_feedCyl:= , 
	HomeLabel_feedCyl:= , 
	WorkLabel_feedCyl:= , 
	HomeSensor_changeCyl:= , 
	WorkSensor_changeCyl:= , 
	HomeValve_changeCyl:= , 
	WorkValve_changeCyl:= , 
	HomeLabel_changeCyl:= , 
	WorkLabel_changeCyl:= , 
	HomeSensor_carrierHold1Cyl:= , 
	WorkSensor_carrierHold1Cyl:= , 
	HomeValve_carrierHold1Cyl:= , 
	WorkValve_carrierHold1Cyl:= , 
	HomeLabel_carrierHold1Cyl:= , 
	WorkLabel_carrierHold1Cyl:= , 
	HomeSensor_carrierHold2Cyl:= , 
	WorkSensor_carrierHold2Cyl:= , 
	HomeValve_carrierHold2Cyl:= , 
	WorkValve_carrierHold2Cyl:= , 
	HomeLabel_carrierHold2Cyl:= , 
	WorkLabel_carrierHold2Cyl:= , 
	HomeSensor_jack3Cyl:= , 
	WorkSensor_jack3Cyl:= , 
	HomeValve_jack3Cyl:= , 
	WorkValve_jack3Cyl:= , 
	HomeLabel_jack3Cyl:= , 
	WorkLabel_jack3Cyl:= , 
	HomeValve_blow:= , 
	WorkValve_blow:= , 
	cableCheckSensor:= , 
	terminalCheckSensor:= , 
	terminalReiveCheckSensor:= , 
	crimpHomeCheckSensor:= , 
	oesReady:= , 
	oesOK:= , 
	HomeSensor_fixCyl:= , 
	WorkSensor_fixCyl:= , 
	HomeValve_fixCyl:= , 
	WorkValve_fixCyl:= , 
	HomeLabel_fixCyl:= , 
	WorkLabel_fixCyl:= , 
	HomeSensor_stepFixCyl:= , 
	WorkSensor_stepFixCyl:= , 
	HomeValve_stepFixCyl:= , 
	WorkValve_stepFixCyl:= , 
	HomeLabel_stepFixCyl:= , 
	WorkLabel_stepFixCyl:= );

END_PROGRAM

// ---- Standard/Module/FAKRA/JacketStripping/FB_JacketStripping_RD.TcPOU
FUNCTION_BLOCK FB_JacketStripping_RD

VAR_IN_OUT
  JacketStripping : UDT_JacketStripping_RD;
  JacketStrippingData : UDT_Data_JacketStripping_RD;  
END_VAR

VAR_INPUT
   //JacketStripping 模组接口
 homeValve_blow : BOOL;
 workValve_blow : BOOL;
 
 homeSensor_gripCyl : BOOL;
 workSensor_gripCyl : BOOL;
 homeValve_gripCyl : BOOL;
 workValve_gripCyl : BOOL;
 homeLabel_gripCyl : STRING[10];
 workLabel_gripCyl : STRING[10];
  
 homeSensor_jackCyl : BOOL;
 workSensor_jackCyl : BOOL;
 homeValve_jackCyl : BOOL;
 workValve_jackCyl : BOOL;
 homeLabel_jackCyl : STRING[10];
 workLabel_jackCyl : STRING[10];
   
 //GS 传送线接口
 homeSensor_fixCyl : BOOL;
 workSensor_fixCyl : BOOL;
 homeValve_fixCyl : BOOL;
 workValve_fixCyl : BOOL;
 homeLabel_fixCyl : STRING[10];
 workLabel_fixCyl : STRING[10];
 
 homeSensor_stepFixCyl : BOOL;
 workSensor_stepFixCyl : BOOL;
 homeValve_stepFixCyl : BOOL;
 workValve_stepFixCyl : BOOL;
 homeLabel_stepFixCyl : STRING[10];
 workLabel_stepFixCyl : STRING[10];
 
END_VAR

VAR  
  machine   : UDT_Machine_RD;
  station   : UDT_Station_RD;
  gripCyl   : UDT_CylinderVar_RD;  
  jackCyl   : UDT_CylinderVar_RD;
  fixCyl    : UDT_CylinderVar_RD;
  stepFixCyl: UDT_CylinderVar_RD;                           
  blow      : UDT_CylinderVar_RD;
  
  rotateAxis    : UDT_AxisVar_RD; 
  cutAxis       : UDT_AxisVar_RD; 
  transferAxis  : UDT_AxisVar_RD; 
  
  badVar :  ARRAY[1..1] OF UDT_BadVar_RD; 
  badData :  ARRAY[1..1] OF UDT_BadData_RD;
  lastProduce : UDT_ProduceDataRecord_RD; 
  produceVari : UDT_ProduceVar_RD; 
  produceData : UDT_ProduceData_RD; 

 
  fB_JacketStripping	: FB_Station_RD;
	fB_gripCyl					: FB_Cylinder_RD;
	fB_jackCyl					: FB_Cylinder_RD;
	fB_fixCyl						: FB_Cylinder_RD;
	fB_stepFixCyl				: FB_Cylinder_RD;
	fB_blow             : FB_Cylinder_RD;
	fb_rotateAxis			  : FB_Axis_RD;
	fb_cutAxis					: FB_Axis_RD;
	fb_transferAxis		  : FB_Axis_RD;
  fb_produce          : FB_Produce_RD;
  
  firstCutTimer :TON;
  firstOpenTimer :TON;
  SecondCutTimer :TON;
  secondOpenTimer :TON;
  blowTimer :TON;
  CommandTimer :TON;
  CommandTime :TIME := T#1S;
  CommandStep : UINT;
  R_Command : R_TRIG;
  
  index : INT; 
  index1 : INT;
  index3 : INT;
  activated : BOOL; 
  tonOn : TON;
  tonOff :TON;
  onePlus : BOOL;
  mcWriteParameterPersistent	: MC_WriteParameterPersistent;	//修改NC参数功能块
  
END_VAR

VAR CONSTANT
  INIT :INT := 0;
  AUTO :INT := 1;
  AUTO2 :INT :=2;
  
  //TransferAxis
  HOME_TRANS        : UINT:=1;
  FIRST_CUT_TRANS		: UINT:=2;
	FIRST_BACK_TRANS	: UINT:=3;
	SECOND_CUT_TRANS	: UINT:=4;
	SECOND_BACK_TRANS	: UINT:=5;
  THIRD_CUT_TRANS	  : UINT:=6;
	THIRD_BACK_TRANS	: UINT:=7;
  FOURTH_CUT_TRANS	: UINT:=8;
	FOURTH_BACK_TRANS	: UINT:=9;
  FIFTH_CUT_TRANS	  : UINT:=10;
	FIFTH_BACK_TRANS	: UINT:=11;

  
  //CutAxis
  HOME_CUT            : UINT:=1;
	FIRST_PRECUT_CUT		: UINT:=2;
	FIRST_CUT_CUT		    : UINT:=3;
	FIRST_BACK_CUT			: UINT:=4;
	SECOND_PRECUT_CUT		: UINT:=5;
	SECOND_CUT_CUT			: UINT:=6;
	SECOND_BACK_CUT			: UINT:=7;
  THIRD_PRECUT_CUT		: UINT:=8;
	THIRD_CUT_CUT		  	: UINT:=9;
	THIRD_BACK_CUT			: UINT:=10;
  FOURTH_PRECUT_CUT		: UINT:=11;
	FOURTH_CUT_CUT		  : UINT:=12;
	FOURTH_BACK_CUT			: UINT:=13;
  FIFTH_PRECUT_CUT		: UINT:=14;
	FIFTH_CUT_CUT	  	  : UINT:=15;
	FIFTH_BACK_CUT			: UINT:=16;  

  //rotateAxis
  HOME_ROTATE   : UINT:=1;

END_VAR

VAR
  
END_VAR

SetUp();
Command();
General();
Permit();
StepInit();
StepAuto();
Alarm();
AutoTip();
ManualTip();
Tip();
Hmi();

ACTION Alarm:
JacketStripping.Message.userAlarms[0] := gripCyl.homeSensorOffAlarm[0];
JacketStripping.Message.userAlarms[1] := gripCyl.homeSensorOnAlarm[0];
JacketStripping.Message.userAlarms[2] := gripCyl.workSensorOffAlarm[0];
JacketStripping.Message.userAlarms[3] := gripCyl.workSensorOnAlarm[0];

JacketStripping.Message.userAlarms[4] := jackCyl.homeSensorOffAlarm[0];
JacketStripping.Message.userAlarms[5] := jackCyl.homeSensorOnAlarm[0];
JacketStripping.Message.userAlarms[6] := jackCyl.workSensorOffAlarm[0];
JacketStripping.Message.userAlarms[7] := jackCyl.workSensorOnAlarm[0];

JacketStripping.Message.userAlarms[8] := fixCyl.homeSensorOffAlarm[0];
JacketStripping.Message.userAlarms[9] := fixCyl.homeSensorOnAlarm[0];
JacketStripping.Message.userAlarms[10] := fixCyl.workSensorOffAlarm[0];
JacketStripping.Message.userAlarms[11] := fixCyl.workSensorOnAlarm[0];

JacketStripping.Message.userAlarms[12] := stepFixCyl.homeSensorOffAlarm[0];
JacketStripping.Message.userAlarms[13] := stepFixCyl.homeSensorOnAlarm[0];
JacketStripping.Message.userAlarms[14] := stepFixCyl.workSensorOffAlarm[0];
JacketStripping.Message.userAlarms[15] := stepFixCyl.workSensorOnAlarm[0];


JacketStripping.Message.userAlarms[16] := rotateAxis.alarming;
JacketStripping.Message.userAlarms[17] := cutAxis.alarming;
JacketStripping.Message.userAlarms[18] := transferAxis.alarming;


JacketStripping.Message.presetAlarms[0] :=station.presetAlarms[0];//工站初始化超时报警

JacketStripping.Message.presetAlarms16 := FUN_AryToWord_RD(JacketStripping.Message.presetAlarms);
JacketStripping.Message.userAlarms64 := FUN_AryToLword_RD(JacketStripping.Message.userAlarms);

(*CASE index OF
    
  0: 
  index1 := 20;
  index := index+10;;
  
  10:
  index1 := index1 +1;
  index := index+10;
  
  20:
  CommandTimer(IN:= FALSE, PT:=CommandTime , Q=> , ET=> );
  JacketStripping.Message.userAlarms[index1] := TRUE;
  index := index+10;

  
  30:
  JacketStripping.Message.userAlarms[index1-1] := FALSE;
  CommandTimer(IN:= TRUE, PT:=CommandTime , Q=> , ET=> );
  IF CommandTimer.Q THEN
    index := index+10;
	END_IF
  
  40:
  IF index1 >=60 THEN
    index := 0;
    ELSIF index1<60 THEN
    index := 10;            
	END_IF
  
	END_CASE*)
END_ACTION

ACTION AutoTip:
JacketStripping.Message.userAutoTips[0] := gripCyl.autoTip ;
JacketStripping.Message.userAutoTips[1] := jackCyl.autoTip ;
JacketStripping.Message.userAutoTips[2] := fixCyl.autoTip ;
JacketStripping.Message.userAutoTips[3] := stepFixCyl.autoTip ;

JacketStripping.Message.userAutoTips[4] := rotateAxis.notPowerOnAutoTip;
JacketStripping.Message.userAutoTips[5] := rotateAxis.notHomeAutoTip;
JacketStripping.Message.userAutoTips[6] := rotateAxis.notInPosAutoTip =HOME_ROTATE;

JacketStripping.Message.userAutoTips[7] := transferAxis.notPowerOnAutoTip;
JacketStripping.Message.userAutoTips[8] := transferAxis.notHomeAutoTip;
JacketStripping.Message.userAutoTips[9] := transferAxis.notInPosAutoTip =HOME_TRANS;
JacketStripping.Message.userAutoTips[10] := transferAxis.notInPosAutoTip =FIRST_CUT_TRANS;
JacketStripping.Message.userAutoTips[11] := transferAxis.notInPosAutoTip =FIRST_BACK_TRANS;
JacketStripping.Message.userAutoTips[12] := transferAxis.notInPosAutoTip =SECOND_CUT_TRANS;
JacketStripping.Message.userAutoTips[13] := transferAxis.notInPosAutoTip =SECOND_BACK_TRANS;
JacketStripping.Message.userAutoTips[14] := transferAxis.notInPosAutoTip =THIRD_CUT_TRANS;
JacketStripping.Message.userAutoTips[15] := transferAxis.notInPosAutoTip =THIRD_BACK_TRANS;
JacketStripping.Message.userAutoTips[16] := transferAxis.notInPosAutoTip =FOURTH_CUT_TRANS;
JacketStripping.Message.userAutoTips[17] := transferAxis.notInPosAutoTip =FOURTH_BACK_TRANS;
JacketStripping.Message.userAutoTips[18] := transferAxis.notInPosAutoTip =FIFTH_CUT_TRANS;
JacketStripping.Message.userAutoTips[19] := transferAxis.notInPosAutoTip =FIFTH_BACK_TRANS;

JacketStripping.Message.userAutoTips[20] := cutAxis.notPowerOnAutoTip;
JacketStripping.Message.userAutoTips[21] := cutAxis.notHomeAutoTip;
JacketStripping.Message.userAutoTips[22] := cutAxis.notInPosAutoTip = HOME_CUT;
JacketStripping.Message.userAutoTips[23] := cutAxis.notInPosAutoTip = FIRST_PRECUT_CUT;
JacketStripping.Message.userAutoTips[24] := cutAxis.notInPosAutoTip = FIRST_CUT_CUT;
JacketStripping.Message.userAutoTips[25] := cutAxis.notInPosAutoTip = FIRST_BACK_CUT;
JacketStripping.Message.userAutoTips[26] := cutAxis.notInPosAutoTip = SECOND_PRECUT_CUT;
JacketStripping.Message.userAutoTips[27] := cutAxis.notInPosAutoTip = SECOND_CUT_CUT;
JacketStripping.Message.userAutoTips[28] := cutAxis.notInPosAutoTip = SECOND_BACK_CUT;
JacketStripping.Message.userAutoTips[29] := cutAxis.notInPosAutoTip = THIRD_PRECUT_CUT;
JacketStripping.Message.userAutoTips[30] := cutAxis.notInPosAutoTip = THIRD_CUT_CUT;
JacketStripping.Message.userAutoTips[31] := cutAxis.notInPosAutoTip = THIRD_BACK_CUT;
JacketStripping.Message.userAutoTips[32] := cutAxis.notInPosAutoTip = FOURTH_PRECUT_CUT;
JacketStripping.Message.userAutoTips[33] := cutAxis.notInPosAutoTip = FOURTH_CUT_CUT;
JacketStripping.Message.userAutoTips[34] := cutAxis.notInPosAutoTip = FOURTH_BACK_CUT	;
JacketStripping.Message.userAutoTips[35] := cutAxis.notInPosAutoTip = FIFTH_PRECUT_CUT;
JacketStripping.Message.userAutoTips[36] := cutAxis.notInPosAutoTip = FIFTH_CUT_CUT;
JacketStripping.Message.userAutoTips[37] := cutAxis.notInPosAutoTip = FIFTH_BACK_CUT;


JacketStripping.Message.presetAutoTips[0] :=   station.presetAutoTips[0]; //工站未初始化
JacketStripping.Message.presetAutoTips[1] :=   station.presetAutoTips[1];   //工站单循环中
JacketStripping.Message.presetAutoTips[2] :=   station.presetAutoTips[2];   //工站运行条件不足

JacketStripping.Message.presetAutoTips16 := FUN_AryToWord_RD(JacketStripping.Message.presetAutoTips);
JacketStripping.Message.userAutoTips64 := FUN_AryToLword_RD(JacketStripping.Message.userAutoTips);
END_ACTION

ACTION Command:
IF activated THEN 
  JacketStripping.UnitState :=ENUM_UnitState.OPERATIONAL;
  ELSE
  JacketStripping.UnitState :=ENUM_UnitState.DISABLED;  
END_IF


IF  station.initDone AND  station.flow[0].actStep = 0  
  AND gripCyl.inHome AND jackCyl.inHome AND blow.inHome AND fixCyl.inHome AND stepFixCyl.inHome 
  AND cutAxis.inPos[HOME_CUT] AND rotateAxis.inPos[HOME_ROTATE] AND transferAxis.inPos[HOME_TRANS] 
 THEN
  JacketStripping.Imm.allObjectInitPos :=TRUE;
  ELSE
   JacketStripping.Imm.allObjectInitPos :=FALSE; 
END_IF



(*R_Command(CLK:= JacketStripping.Command <> 0 AND JacketStripping.CommandState = ENUM_ExecState.READY, Q=>);

CASE CommandStep OF

0: IF JacketStripping.Command =ENUM_StationCommand.INIT AND R_Command.Q THEN CommandStep := 100;
   ELSIF JacketStripping.Command =ENUM_StationCommand.START AND R_Command.Q THEN  CommandStep := 200;
   ELSIF JacketStripping.Command =ENUM_StationCommand.STOP AND R_Command.Q THEN  CommandStep := 300;  
   END_IF

END_CASE*)
END_ACTION

ACTION General:
IF machine.reset THEN 
  machine.tipReset := TRUE ;
  MEMSET(destAddr:=ADR(machine.presetManualTips) , fillByte:= 0, n:=SIZEOF(machine.presetManualTips));
 ELSE
  machine.tipReset := FALSE ;
END_IF
END_ACTION

ACTION Hmi:
// 触摸屏弹窗

JacketStripping.Message.popupTrigger.1 := 
  JacketStripping.Message.presetManualTips16 <> 0 OR 
  JacketStripping.Message.userManualTips64<> 0;
  
JacketStripping.Message.popupTrigger.2 :=
(JacketStripping.Message.presetAutoTips16 <> 0 OR 
JacketStripping.Message.userAutoTips64 <> 0) AND 
(station.autoTipTrigger OR machine.autoMode) ;

IF machine.reset THEN
  machine.popup:= 0;
END_IF

//.0 alarmTrigger 
//.1 manualTipTrigger
//.2 autoTipTrigger
//.3 tipTrigger

gripCyl.homehmi:=JacketStripping.Hmi.gripCyl.homehmi;// 原点hmi
JacketStripping.Hmi.gripCyl.homeForbidIcon:=gripCyl.homeForbidIcon;// 原点禁止图标
JacketStripping.Hmi.gripCyl.homeValve:=gripCyl.homeValve;// 原点阀
JacketStripping.Hmi.gripCyl.homeManual:=gripCyl.homeManual;// 原点Manual
gripCyl.workhmi:=JacketStripping.Hmi.gripCyl.workhmi;// 动点hmi
JacketStripping.Hmi.gripCyl.workForbidIcon:=gripCyl.workForbidIcon;// 动点禁止图标
JacketStripping.Hmi.gripCyl.workValve:=gripCyl.workValve;// 动点阀
JacketStripping.Hmi.gripCyl.workManual:=gripCyl.workManual;// 动点Manual
JacketStripping.Hmi.gripCyl.homeSensor[0]:=gripCyl.homeSensor[0];// 原点传感器
JacketStripping.Hmi.gripCyl.workSensor[0]:=gripCyl.workSensor[0];// 动点传感器
JacketStripping.Hmi.gripCyl.homeSensorLabel[0]:=gripCyl.homeSensorLabel[0];// 原点传感器标签
JacketStripping.Hmi.gripCyl.workSensorLabel[0]:=gripCyl.workSensorLabel[0];// 动点传感器标签
JacketStripping.Hmi.gripCyl.toHomeActionTime:=gripCyl.toHomeActionTime;// 到原点所用时间
JacketStripping.Hmi.gripCyl.toWorkActionTime:=gripCyl.toWorkActionTime;// 到动点所用时间


jackCyl.homehmi:=JacketStripping.Hmi.jackCyl.homehmi;// 原点hmi
JacketStripping.Hmi.jackCyl.homeForbidIcon:=jackCyl.homeForbidIcon;// 原点禁止图标
JacketStripping.Hmi.jackCyl.homeValve:=jackCyl.homeValve;// 原点阀
JacketStripping.Hmi.jackCyl.homeManual:=jackCyl.homeManual;// 原点Manual
jackCyl.workhmi:=JacketStripping.Hmi.jackCyl.workhmi;// 动点hmi
JacketStripping.Hmi.jackCyl.workForbidIcon:=jackCyl.workForbidIcon;// 动点禁止图标
JacketStripping.Hmi.jackCyl.workValve:=jackCyl.workValve;// 动点阀
JacketStripping.Hmi.jackCyl.workManual:=jackCyl.workManual;// 动点Manual
JacketStripping.Hmi.jackCyl.homeSensor[0]:=jackCyl.homeSensor[0];// 原点传感器
JacketStripping.Hmi.jackCyl.workSensor[0]:=jackCyl.workSensor[0];// 动点传感器
JacketStripping.Hmi.jackCyl.homeSensorLabel[0]:=jackCyl.homeSensorLabel[0];// 原点传感器标签
JacketStripping.Hmi.jackCyl.workSensorLabel[0]:=jackCyl.workSensorLabel[0];// 动点传感器标签
JacketStripping.Hmi.jackCyl.toHomeActionTime:=jackCyl.toHomeActionTime;// 到原点所用时间
JacketStripping.Hmi.jackCyl.toWorkActionTime:=jackCyl.toWorkActionTime;// 到动点所用时间


fixCyl.homehmi:=JacketStripping.Hmi.fixCyl.homehmi;// 原点hmi
JacketStripping.Hmi.fixCyl.homeForbidIcon:=fixCyl.homeForbidIcon;// 原点禁止图标
JacketStripping.Hmi.fixCyl.homeValve:=fixCyl.homeValve;// 原点阀
JacketStripping.Hmi.fixCyl.homeManual:=fixCyl.homeManual;// 原点Manual
fixCyl.workhmi:=JacketStripping.Hmi.fixCyl.workhmi;// 动点hmi
JacketStripping.Hmi.fixCyl.workForbidIcon:=fixCyl.workForbidIcon;// 动点禁止图标
JacketStripping.Hmi.fixCyl.workValve:=fixCyl.workValve;// 动点阀
JacketStripping.Hmi.fixCyl.workManual:=fixCyl.workManual;// 动点Manual
JacketStripping.Hmi.fixCyl.homeSensor[0]:=fixCyl.homeSensor[0];// 原点传感器
JacketStripping.Hmi.fixCyl.workSensor[0]:=fixCyl.workSensor[0];// 动点传感器
JacketStripping.Hmi.fixCyl.homeSensorLabel[0]:=fixCyl.homeSensorLabel[0];// 原点传感器标签
JacketStripping.Hmi.fixCyl.workSensorLabel[0]:=fixCyl.workSensorLabel[0];// 动点传感器标签
JacketStripping.Hmi.fixCyl.toHomeActionTime:=fixCyl.toHomeActionTime;// 到原点所用时间
JacketStripping.Hmi.fixCyl.toWorkActionTime:=fixCyl.toWorkActionTime;// 到动点所用时间


stepFixCyl.homehmi:=JacketStripping.Hmi.stepFixCyl.homehmi;// 原点hmi
JacketStripping.Hmi.stepFixCyl.homeForbidIcon:=stepFixCyl.homeForbidIcon;// 原点禁止图标
JacketStripping.Hmi.stepFixCyl.homeValve:=stepFixCyl.homeValve;// 原点阀
JacketStripping.Hmi.stepFixCyl.homeManual:=stepFixCyl.homeManual;// 原点Manual
stepFixCyl.workhmi:=JacketStripping.Hmi.stepFixCyl.workhmi;// 动点hmi
JacketStripping.Hmi.stepFixCyl.workForbidIcon:=stepFixCyl.workForbidIcon;// 动点禁止图标
JacketStripping.Hmi.stepFixCyl.workValve:=stepFixCyl.workValve;// 动点阀
JacketStripping.Hmi.stepFixCyl.workManual:=stepFixCyl.workManual;// 动点Manual
JacketStripping.Hmi.stepFixCyl.homeSensor[0]:=stepFixCyl.homeSensor[0];// 原点传感器
JacketStripping.Hmi.stepFixCyl.workSensor[0]:=stepFixCyl.workSensor[0];// 动点传感器
JacketStripping.Hmi.stepFixCyl.homeSensorLabel[0]:=stepFixCyl.homeSensorLabel[0];// 原点传感器标签
JacketStripping.Hmi.stepFixCyl.workSensorLabel[0]:=stepFixCyl.workSensorLabel[0];// 动点传感器标签
JacketStripping.Hmi.stepFixCyl.toHomeActionTime:=stepFixCyl.toHomeActionTime;// 到原点所用时间
JacketStripping.Hmi.stepFixCyl.toWorkActionTime:=stepFixCyl.toWorkActionTime;// 到动点所用时间


blow.homehmi:=JacketStripping.Hmi.blow.homehmi;// 原点hmi
JacketStripping.Hmi.blow.homeForbidIcon:=blow.homeForbidIcon;// 原点禁止图标
JacketStripping.Hmi.blow.homeValve:=blow.homeValve;// 原点阀
JacketStripping.Hmi.blow.homeManual:=blow.homeManual;// 原点Manual
blow.workhmi:=JacketStripping.Hmi.blow.workhmi;// 动点hmi
JacketStripping.Hmi.blow.workForbidIcon:=blow.workForbidIcon;// 动点禁止图标
JacketStripping.Hmi.blow.workValve:=blow.workValve;// 动点阀
JacketStripping.Hmi.blow.workManual:=blow.workManual;// 动点Manual
JacketStripping.Hmi.blow.homeSensor[0]:=blow.homeSensor[0];// 原点传感器
JacketStripping.Hmi.blow.workSensor[0]:=blow.workSensor[0];// 动点传感器
JacketStripping.Hmi.blow.homeSensorLabel[0]:=blow.homeSensorLabel[0];// 原点传感器标签
JacketStripping.Hmi.blow.workSensorLabel[0]:=blow.workSensorLabel[0];// 动点传感器标签
JacketStripping.Hmi.blow.toHomeActionTime:=blow.toHomeActionTime;// 到原点所用时间
JacketStripping.Hmi.blow.toWorkActionTime:=blow.toWorkActionTime;// 到动点所用时间


rotateAxis.powerhmi:=JacketStripping.Hmi.rotateAxis.powerhmi;// 伺服Onhmi
JacketStripping.Hmi.rotateAxis.powerForbidIcon:=rotateAxis.powerForbidIcon;// 伺服On禁止图标
JacketStripping.Hmi.rotateAxis.isPowerOn:=rotateAxis.isPowerOn;// 伺服On状态
rotateAxis.halthmi:=JacketStripping.Hmi.rotateAxis.halthmi;// 伺服暂停hmi
rotateAxis.resethmi:=JacketStripping.Hmi.rotateAxis.resethmi;// 伺服复位hmi
rotateAxis.jogForwardhmi:=JacketStripping.Hmi.rotateAxis.jogForwardhmi;// 伺服JOG+_hmi
JacketStripping.Hmi.rotateAxis.jogForwardForbidIcon:=rotateAxis.jogForwardForbidIcon;// 伺服JOG+禁止图标
rotateAxis.jogBackwardshmi:=JacketStripping.Hmi.rotateAxis.jogBackwardshmi;// 伺服JOG-hmi
JacketStripping.Hmi.rotateAxis.jogBackwardsForbidIcon:=rotateAxis.jogBackwardsForbidIcon;// 伺服JOG-禁止图标
rotateAxis.homehmi:=JacketStripping.Hmi.rotateAxis.homehmi;// 伺服回原点hmi
JacketStripping.Hmi.rotateAxis.homeForbidIcon:=rotateAxis.homeForbidIcon;// 伺服回原点禁止图标
JacketStripping.Hmi.rotateAxis.homeDone:=rotateAxis.homeDone;// 伺服回原点完成
rotateAxis.brakehmi:=JacketStripping.Hmi.rotateAxis.brakehmi;// 伺服刹车hmi
JacketStripping.Hmi.rotateAxis.brakeForbidIcon:=rotateAxis.brakeForbidIcon;// 伺服刹车禁止图标
JacketStripping.Hmi.rotateAxis.brake:=rotateAxis.brake;// 伺服刹车输出
rotateAxis.movehmi:=JacketStripping.Hmi.rotateAxis.movehmi;// 定位启动hmi
JacketStripping.Hmi.rotateAxis.moveForbidIcon:=rotateAxis.moveForbidIcon;// 定位启动禁止图标
rotateAxis.posTeach:=JacketStripping.Hmi.rotateAxis.posTeach;// 当前位置示教
rotateAxis.movehmiNo:=JacketStripping.Hmi.rotateAxis.movehmiNo;// 手动定位编号
JacketStripping.Hmi.rotateAxis.inPosNo:=rotateAxis.inPosNo;// 伺服到位编号
JacketStripping.Hmi.rotateAxis.status:=rotateAxis.status;// 伺服状态
JacketStripping.Hmi.rotateAxis.ncErrID:=rotateAxis.ncErrID;// 伺服NC错误代码
JacketStripping.Hmi.rotateAxis.warnID :=rotateAxis.warnID ;// 伺服警告代码
JacketStripping.Hmi.rotateAxis.driverErrID:=rotateAxis.driverErrID;// 伺服驱动器代码
JacketStripping.Hmi.rotateAxis.posUnit:=rotateAxis.posUnit;// 位置单位
JacketStripping.Hmi.rotateAxis.veloUnit:=rotateAxis.veloUnit;// 速度单位
JacketStripping.Hmi.rotateAxis.accDecUnit:=rotateAxis.accDecUnit;// 加/减速度单位
JacketStripping.Hmi.rotateAxis.actPos:=rotateAxis.actPos;// 当前坐标
JacketStripping.Hmi.rotateAxis.actVelo:=rotateAxis.actVelo;// 当前速度
JacketStripping.Hmi.rotateAxis.actTorque:=rotateAxis.actTorque;// 当前转矩
JacketStripping.Hmi.rotateAxis.lsp:=rotateAxis.lsp;// 伺服正极限
JacketStripping.Hmi.rotateAxis.lsn:=rotateAxis.lsn;// 伺服负极限
JacketStripping.Hmi.rotateAxis.dog:=rotateAxis.dog;// 伺服原点感应
JacketStripping.Hmi.rotateAxis.targetDistance:=rotateAxis.targetDistance;// 目标距离
JacketStripping.Hmi.rotateAxis.targetVelocity:=rotateAxis.targetVelocity;// 目标速度





cutAxis.powerhmi:=JacketStripping.Hmi.cutAxis.powerhmi;// 伺服Onhmi
JacketStripping.Hmi.cutAxis.powerForbidIcon:=cutAxis.powerForbidIcon;// 伺服On禁止图标
JacketStripping.Hmi.cutAxis.isPowerOn:=cutAxis.isPowerOn;// 伺服On状态
cutAxis.halthmi:=JacketStripping.Hmi.cutAxis.halthmi;// 伺服暂停hmi
cutAxis.resethmi:=JacketStripping.Hmi.cutAxis.resethmi;// 伺服复位hmi
cutAxis.jogForwardhmi:=JacketStripping.Hmi.cutAxis.jogForwardhmi;// 伺服JOG+_hmi
JacketStripping.Hmi.cutAxis.jogForwardForbidIcon:=cutAxis.jogForwardForbidIcon;// 伺服JOG+禁止图标
cutAxis.jogBackwardshmi:=JacketStripping.Hmi.cutAxis.jogBackwardshmi;// 伺服JOG-hmi
JacketStripping.Hmi.cutAxis.jogBackwardsForbidIcon:=cutAxis.jogBackwardsForbidIcon;// 伺服JOG-禁止图标
cutAxis.homehmi:=JacketStripping.Hmi.cutAxis.homehmi;// 伺服回原点hmi
JacketStripping.Hmi.cutAxis.homeForbidIcon:=cutAxis.homeForbidIcon;// 伺服回原点禁止图标
JacketStripping.Hmi.cutAxis.homeDone:=cutAxis.homeDone;// 伺服回原点完成
cutAxis.brakehmi:=JacketStripping.Hmi.cutAxis.brakehmi;// 伺服刹车hmi
JacketStripping.Hmi.cutAxis.brakeForbidIcon:=cutAxis.brakeForbidIcon;// 伺服刹车禁止图标
JacketStripping.Hmi.cutAxis.brake:=cutAxis.brake;// 伺服刹车输出
cutAxis.movehmi:=JacketStripping.Hmi.cutAxis.movehmi;// 定位启动hmi
JacketStripping.Hmi.cutAxis.moveForbidIcon:=cutAxis.moveForbidIcon;// 定位启动禁止图标
cutAxis.posTeach:=JacketStripping.Hmi.cutAxis.posTeach;// 当前位置示教
cutAxis.movehmiNo:=JacketStripping.Hmi.cutAxis.movehmiNo;// 手动定位编号
JacketStripping.Hmi.cutAxis.inPosNo:=cutAxis.inPosNo;// 伺服到位编号
JacketStripping.Hmi.cutAxis.status:=cutAxis.status;// 伺服状态
JacketStripping.Hmi.cutAxis.ncErrID:=cutAxis.ncErrID;// 伺服NC错误代码
JacketStripping.Hmi.cutAxis.driverErrID:=cutAxis.driverErrID;// 伺服驱动器代码
JacketStripping.Hmi.cutAxis.warnID :=cutAxis.warnID ;// 伺服警告代码
JacketStripping.Hmi.cutAxis.posUnit:=cutAxis.posUnit;// 位置单位
JacketStripping.Hmi.cutAxis.veloUnit:=cutAxis.veloUnit;// 速度单位
JacketStripping.Hmi.cutAxis.accDecUnit:=cutAxis.accDecUnit;// 加/减速度单位
JacketStripping.Hmi.cutAxis.actPos:=cutAxis.actPos;// 当前坐标
JacketStripping.Hmi.cutAxis.actVelo:=cutAxis.actVelo;// 当前速度
JacketStripping.Hmi.cutAxis.actTorque:=cutAxis.actTorque;// 当前转矩
JacketStripping.Hmi.cutAxis.lsp:=cutAxis.lsp;// 伺服正极限
JacketStripping.Hmi.cutAxis.lsn:=cutAxis.lsn;// 伺服负极限
JacketStripping.Hmi.cutAxis.dog:=cutAxis.dog;// 伺服原点感应
JacketStripping.Hmi.cutAxis.targetDistance:=cutAxis.targetDistance;// 目标距离
JacketStripping.Hmi.cutAxis.targetVelocity:=cutAxis.targetVelocity;// 目标速度




transferAxis.powerhmi:=JacketStripping.Hmi.transferAxis.powerhmi;// 伺服Onhmi
JacketStripping.Hmi.transferAxis.powerForbidIcon:=transferAxis.powerForbidIcon;// 伺服On禁止图标
JacketStripping.Hmi.transferAxis.isPowerOn:=transferAxis.isPowerOn;// 伺服On状态
transferAxis.halthmi:=JacketStripping.Hmi.transferAxis.halthmi;// 伺服暂停hmi
transferAxis.resethmi:=JacketStripping.Hmi.transferAxis.resethmi;// 伺服复位hmi
transferAxis.jogForwardhmi:=JacketStripping.Hmi.transferAxis.jogForwardhmi;// 伺服JOG+_hmi
JacketStripping.Hmi.transferAxis.jogForwardForbidIcon:=transferAxis.jogForwardForbidIcon;// 伺服JOG+禁止图标
transferAxis.jogBackwardshmi:=JacketStripping.Hmi.transferAxis.jogBackwardshmi;// 伺服JOG-hmi
JacketStripping.Hmi.transferAxis.jogBackwardsForbidIcon:=transferAxis.jogBackwardsForbidIcon;// 伺服JOG-禁止图标
transferAxis.homehmi:=JacketStripping.Hmi.transferAxis.homehmi;// 伺服回原点hmi
JacketStripping.Hmi.transferAxis.homeForbidIcon:=transferAxis.homeForbidIcon;// 伺服回原点禁止图标
JacketStripping.Hmi.transferAxis.homeDone:=transferAxis.homeDone;// 伺服回原点完成
transferAxis.brakehmi:=JacketStripping.Hmi.transferAxis.brakehmi;// 伺服刹车hmi
JacketStripping.Hmi.transferAxis.brakeForbidIcon:=transferAxis.brakeForbidIcon;// 伺服刹车禁止图标
JacketStripping.Hmi.transferAxis.brake:=transferAxis.brake;// 伺服刹车输出
transferAxis.movehmi:=JacketStripping.Hmi.transferAxis.movehmi;// 定位启动hmi
JacketStripping.Hmi.transferAxis.moveForbidIcon:=transferAxis.moveForbidIcon;// 定位启动禁止图标
transferAxis.posTeach:=JacketStripping.Hmi.transferAxis.posTeach;// 当前位置示教
transferAxis.movehmiNo:=JacketStripping.Hmi.transferAxis.movehmiNo;// 手动定位编号
JacketStripping.Hmi.transferAxis.inPosNo:=transferAxis.inPosNo;// 伺服到位编号
JacketStripping.Hmi.transferAxis.status:=transferAxis.status;// 伺服状态
JacketStripping.Hmi.transferAxis.ncErrID:=transferAxis.ncErrID;// 伺服NC错误代码
JacketStripping.Hmi.transferAxis.driverErrID:=transferAxis.driverErrID;// 伺服驱动器代码
JacketStripping.Hmi.transferAxis.warnID :=transferAxis.warnID ;// 伺服警告代码
JacketStripping.Hmi.transferAxis.posUnit:=transferAxis.posUnit;// 位置单位
JacketStripping.Hmi.transferAxis.veloUnit:=transferAxis.veloUnit;// 速度单位
JacketStripping.Hmi.transferAxis.accDecUnit:=transferAxis.accDecUnit;// 加/减速度单位
JacketStripping.Hmi.transferAxis.actPos:=transferAxis.actPos;// 当前坐标
JacketStripping.Hmi.transferAxis.actVelo:=transferAxis.actVelo;// 当前速度
JacketStripping.Hmi.transferAxis.actTorque:=transferAxis.actTorque;// 当前转矩
JacketStripping.Hmi.transferAxis.lsp:=transferAxis.lsp;// 伺服正极限
JacketStripping.Hmi.transferAxis.lsn:=transferAxis.lsn;// 伺服负极限
JacketStripping.Hmi.transferAxis.dog:=transferAxis.dog;// 伺服原点感应
JacketStripping.Hmi.transferAxis.targetDistance:=transferAxis.targetDistance;// 目标距离
JacketStripping.Hmi.transferAxis.targetVelocity:=transferAxis.targetVelocity;// 目标速度


Station.inithmi:=JacketStripping.Hmi.Station.inithmi;// 工站初始化hmi
JacketStripping.Hmi.Station.initForbidIcon:=Station.initForbidIcon;// 工站初始化禁止图标
JacketStripping.Hmi.Station.initing:=Station.initing;// 工站初始化中
Station.cycleRunhmi:=JacketStripping.Hmi.Station.cycleRunhmi;// 工站单循环hmi
JacketStripping.Hmi.Station.cycleRunForbidIcon:=Station.cycleRunForbidIcon;// 工站单循环禁止图标
JacketStripping.Hmi.Station.cycleRunning:=Station.cycleRunning;// 工站单循环中
Station.jogRunhmi:=JacketStripping.Hmi.Station.jogRunhmi;// 工站寸动hmi
JacketStripping.Hmi.Station.jogRunForbidIcon:=Station.jogRunForbidIcon;// 工站寸动禁止图标
JacketStripping.Hmi.Station.jogRunning:=Station.jogRunning;// 工站寸动中
Station.pausehmi:=JacketStripping.Hmi.Station.pausehmi;// 工站暂停hmi
Station.disablehmi:=JacketStripping.Hmi.Station.disablehmi;// 工站屏蔽hmi
Station.repetitionsEnable:=JacketStripping.Hmi.Station.repetitionsEnable;// 单循环重复动作开启
Station.repetitionsClear:=JacketStripping.Hmi.Station.repetitionsClear;// 单循环重复动作计数清零
JacketStripping.Hmi.Station.repetitions:=Station.repetitions;// 单循环重复动作计数
Station.repetitionsTimes:=JacketStripping.Hmi.Station.repetitionsTimes;// 单循环重复动作次数设置
JacketStripping.Hmi.Station.status:=Station.status;// 工站状态显示
JacketStripping.Hmi.Station.cycleTime:=Station.cycleTime;// 工站周期时间
JacketStripping.Hmi.Station.flow[0].actStep:=Station.flow[0].actStep;// 流程当前步号
JacketStripping.Hmi.Station.flow[1].actStep:=Station.flow[1].actStep;// 流程当前步号
END_ACTION

ACTION ManualTip:
 JacketStripping.Message.presetManualTips[0] := machine.presetManualTips[0];//急停中,无法操作
 JacketStripping.Message.presetManualTips[1] := machine.presetManualTips[1];//安全条件不满足,无法操作
 JacketStripping.Message.presetManualTips[2] := machine.presetManualTips[2];//安全门未锁好,无法操作
 JacketStripping.Message.presetManualTips[3] := machine.presetManualTips[3];//气压不足,无法操作
 JacketStripping.Message.presetManualTips[4] := machine.presetManualTips[4];//不在手动模式,无法操作
 
 JacketStripping.Message.userManualTips[0]:= rotateAxis.notPowerOnManualTip;
 JacketStripping.Message.userManualTips[1]:= rotateAxis.unableBrakeManualTip;
 JacketStripping.Message.userManualTips[2]:= rotateAxis.unablePowerOnManualTip;
 JacketStripping.Message.userManualTips[3]:= cutAxis.notPowerOnManualTip;
 JacketStripping.Message.userManualTips[4]:= cutAxis.unableBrakeManualTip;
 JacketStripping.Message.userManualTips[5]:= cutAxis.unablePowerOnManualTip;
 JacketStripping.Message.userManualTips[6]:= transferAxis.notPowerOnManualTip;
 JacketStripping.Message.userManualTips[7]:= transferAxis.unableBrakeManualTip;
 JacketStripping.Message.userManualTips[8]:= transferAxis.unablePowerOnManualTip;
 JacketStripping.Message.userManualTips[9]:= fixCyl.noWorkPermitManualTip;
 JacketStripping.Message.userManualTips[10]:= stepFixCyl.noWorkPermitManualTip;
 
 
 JacketStripping.Message.presetManualTips16 := FUN_AryToWord_RD(JacketStripping.Message.presetManualTips);
 JacketStripping.Message.userManualTips64 := FUN_AryToLword_RD(JacketStripping.Message.userManualTips);
END_ACTION

ACTION Permit:
fixCyl.workPermit := JacketStripping.Imm.carrierInPos;
stepFixCyl.workPermit := JacketStripping.Imm.carrierInPos;
JacketStripping.Imm.carrierFree := gripCyl.inHome AND jackCyl.inHome  AND fixCyl.inHome AND stepFixCyl.inHome AND transferAxis.inPos[HOME_TRANS];
END_ACTION

ACTION SetUp:
//FB

  fb_JacketStripping(machine:=Machine , station:=station );
  
  fb_gripCyl(machine:= Machine, station:= station, vari:= gripCyl, data:=JacketStrippingData.GripCyl );
  fb_jackCyl(machine:=Machine , station:=station , vari:= jackCyl, data:= JacketStrippingData.JackCyl);
  fb_blow(machine:= Machine, station:= station, vari:=blow , data:= JacketStrippingData.Blow);
  
  fb_fixCyl(machine:= Machine, station:= station, vari:= fixCyl, data:=JacketStrippingData.FixCyl );
  fb_stepFixCyl(machine:=Machine , station:=station , vari:= stepFixCyl, data:=JacketStrippingData.StepFixCyl );
  
  fb_rotateAxis(machine:= Machine, station:= station, vari:= rotateAxis, data:= JacketStrippingData.RotateAxis);
  fb_transferAxis(machine:= Machine, station:= station, vari:= transferAxis, data:= JacketStrippingData.TransferAxis);
  fb_cutAxis(machine:= Machine, station:= station, vari:= cutAxis, data:= JacketStrippingData.CutAxis);
   
  fb_produce(machine:= Machine, station:= station, vari:= produceVari, data:= produceData, badVar:= badVar, badData:= badData, lastProduce:=lastProduce );
  

//Imm

  Machine.airOn := JacketStripping.Imm.Machine_airOn;
  Machine.allDoorClosed:=JacketStripping.Imm.Machine_allDoorClosed;
  Machine.eStop:=JacketStripping.Imm.Machine_eStop;
  Machine.safety:=JacketStripping.Imm.Machine_safety;
  Machine.manualMode:=JacketStripping.Imm.Machine_manualMode;
  Machine.autoMode:=JacketStripping.Imm.Machine_autoMode;
  Machine.reset := JacketStripping.Imm.Machine_reset;
  machine.stopping := JacketStripping.Imm.Machine_stopping;

  
   
  station.canRun:= JacketStripping.Imm.stationCanRun; 
  station.done := JacketStripping.Imm.stationDone;
 
// VAR INPUT
  
